LIN {X 0,Y 573.242,Z 122.078,A -85,B 0,C 180,E1 -2301.298,E2 -2301.298} C_VEL
LIN {X 0,Y 573.212,Z 122.081,A -85,B 0,C 180,E1 -2304.018,E2 -2304.018} C_VEL
LIN {X 0,Y 573.238,Z 122.074,A -85,B 0,C 180,E1 -2306.515,E2 -2306.515} C_VEL
LIN {X 0,Y 573.224,Z 122.08,A -85,B 0,C 180,E1 -2309.118,E2 -2309.118} C_VEL
LIN {X 0,Y 573.251,Z 122.075,A -85,B 0,C 180,E1 -2311.971,E2 -2311.971} C_VEL
LIN {X 0,Y 573.252,Z 122.073,A -85,B 0,C 180,E1 -2314.589,E2 -2314.589} C_VEL
LIN {X 0,Y 573.236,Z 122.079,A -85,B 0,C 180,E1 -2317.662,E2 -2317.662} C_VEL
LIN {X 0,Y 573.265,Z 122.073,A -85,B 0,C 180,E1 -2320.67,E2 -2320.67} C_VEL
LIN {X 0,Y 573.246,Z 122.076,A -85,B 0,C 180,E1 -2323.621,E2 -2323.621} C_VEL
LIN {X 0,Y 573.272,Z 122.071,A -85,B 0,C 180,E1 -2325.807,E2 -2325.807} C_VEL
LIN {X 0,Y 573.262,Z 122.076,A -85,B 0,C 180,E1 -2328.745,E2 -2328.745} C_VEL
LIN {X 0,Y 573.281,Z 122.071,A -85,B 0,C 180,E1 -2331.54,E2 -2331.54} C_VEL
LIN {X 0,Y 573.298,Z 122.069,A -85,B 0,C 180,E1 -2334.372,E2 -2334.372} C_VEL
LIN {X 0,Y 573.313,Z 122.065,A -85,B 0,C 180,E1 -2337.892,E2 -2337.892} C_VEL
LIN {X 0,Y 573.334,Z 122.07,A -85,B 0,C 180,E1 -2340.702,E2 -2340.702} C_VEL
LIN {X 0,Y 573.305,Z 122.076,A -85,B 0,C 180,E1 -2342.81,E2 -2342.81} C_VEL
LIN {X 0,Y 573.294,Z 122.067,A -85,B 0,C 180,E1 -2345.628,E2 -2345.628} C_VEL
LIN {X 0,Y 573.289,Z 122.074,A -85,B 0,C 180,E1 -2348.459,E2 -2348.459} C_VEL
LIN {X 0,Y 573.27,Z 122.071,A -85,B 0,C 180,E1 -2351.312,E2 -2351.312} C_VEL
LIN {X 0,Y 573.27,Z 122.074,A -85,B 0,C 180,E1 -2354.193,E2 -2354.193} C_VEL
LIN {X 0,Y 573.256,Z 122.074,A -85,B 0,C 180,E1 -2357.111,E2 -2357.111} C_VEL
LIN {X 0,Y 573.25,Z 122.077,A -85,B 0,C 180,E1 -2360.076,E2 -2360.076} C_VEL
LIN {X 0,Y 573.231,Z 122.076,A -85,B 0,C 180,E1 -2363.099,E2 -2363.099} C_VEL
LIN {X 0,Y 573.247,Z 122.076,A -85,B 0,C 180,E1 -2364.39,E2 -2364.39} C_VEL
LIN {X 0,Y 572.622,Z 122.156,A -85,B 0,C 180,E1 -2364.976,E2 -2364.976} C_VEL
LIN {X 0,Y 569.783,Z 122.509,A -85,B 0,C 180,E1 -2365.928,E2 -2365.928} C_VEL
LIN {X 0,Y 567.355,Z 122.811,A -85,B 0,C 180,E1 -2366.694,E2 -2366.694} C_VEL
LIN {X 0,Y 566.303,Z 122.939,A -85,B 0,C 180,E1 -2367.285,E2 -2367.285} C_VEL
LIN {X 0,Y 566.214,Z 122.95,A -85,B 0,C 180,E1 -2367.485,E2 -2367.485} C_VEL
LIN {X 0,Y 566.184,Z 122.957,A -85,B 0,C 180,E1 -2370.592,E2 -2370.592} C_VEL
LIN {X 0,Y 566.225,Z 122.948,A -85,B 0,C 180,E1 -2373.101,E2 -2373.101} C_VEL
LIN {X 0,Y 566.211,Z 122.958,A -85,B 0,C 180,E1 -2376.216,E2 -2376.216} C_VEL
LIN {X 0,Y 566.219,Z 122.949,A -85,B 0,C 180,E1 -2379.273,E2 -2379.273} C_VEL
LIN {X 0,Y 566.21,Z 122.958,A -85,B 0,C 180,E1 -2382.087,E2 -2382.087} C_VEL
LIN {X 0,Y 566.169,Z 122.955,A -85,B 0,C 180,E1 -2385.036,E2 -2385.036} C_VEL
LIN {X 0,Y 566.21,Z 122.959,A -85,B 0,C 180,E1 -2387.913,E2 -2387.913} C_VEL
LIN {X 0,Y 566.218,Z 122.949,A -85,B 0,C 180,E1 -2390.727,E2 -2390.727} C_VEL
LIN {X 0,Y 566.202,Z 122.96,A -85,B 0,C 180,E1 -2393.785,E2 -2393.785} C_VEL
LIN {X 0,Y 566.225,Z 122.948,A -85,B 0,C 180,E1 -2396.899,E2 -2396.899} C_VEL
LIN {X 0,Y 566.184,Z 122.959,A -85,B 0,C 180,E1 -2399.408,E2 -2399.408} C_VEL
LIN {X 0,Y 566.224,Z 122.953,A -85,B 0,C 180,E1 -2401.858,E2 -2401.858} C_VEL
LIN {X 0,Y 566.211,Z 122.95,A -85,B 0,C 180,E1 -2404.251,E2 -2404.251} C_VEL
LIN {X 0,Y 566.187,Z 122.953,A -85,B 0,C 180,E1 -2406.714,E2 -2406.714} C_VEL
LIN {X 0,Y 566.214,Z 122.955,A -85,B 0,C 180,E1 -2409.663,E2 -2409.663} C_VEL
LIN {X 0,Y 566.196,Z 122.953,A -85,B 0,C 180,E1 -2412.669,E2 -2412.669} C_VEL
LIN {X 0,Y 566.23,Z 122.952,A -85,B 0,C 180,E1 -2415.627,E2 -2415.627} C_VEL
LIN {X 0,Y 566.231,Z 122.949,A -85,B 0,C 180,E1 -2418.675,E2 -2418.675} C_VEL
LIN {X 0,Y 566.23,Z 122.953,A -85,B 0,C 180,E1 -2421.435,E2 -2421.435} C_VEL
LIN {X 0,Y 566.266,Z 122.943,A -85,B 0,C 180,E1 -2424.302,E2 -2424.302} C_VEL
LIN {X 0,Y 566.284,Z 122.941,A -85,B 0,C 180,E1 -2427.867,E2 -2427.867} C_VEL
LIN {X 0,Y 566.3,Z 122.944,A -85,B 0,C 180,E1 -2430.711,E2 -2430.711} C_VEL
LIN {X 0,Y 566.269,Z 122.951,A -85,B 0,C 180,E1 -2432.846,E2 -2432.846} C_VEL
LIN {X 0,Y 566.266,Z 122.943,A -85,B 0,C 180,E1 -2435.699,E2 -2435.699} C_VEL
LIN {X 0,Y 566.231,Z 122.953,A -85,B 0,C 180,E1 -2438.566,E2 -2438.566} C_VEL
LIN {X 0,Y 566.24,Z 122.947,A -85,B 0,C 180,E1 -2441.455,E2 -2441.455} C_VEL
LIN {X 0,Y 566.232,Z 122.954,A -85,B 0,C 180,E1 -2444.507,E2 -2444.507} C_VEL
LIN {X 0,Y 566.198,Z 122.954,A -85,B 0,C 180,E1 -2447.332,E2 -2447.332} C_VEL
LIN {X 0,Y 566.25,Z 123.012,A -85,B 0,C 180,E1 -2449.58,E2 -2449.58} C_VEL
LIN {X 0,Y 566.372,Z 130.978,A -85,B 0,C 180,E1 -2451.092,E2 -2451.092} C_VEL
LIN {X 0,Y 566.202,Z 146.316,A -85,B 0,C 180,E1 -2453.986,E2 -2453.986} C_VEL
LIN {X 0,Y 566.206,Z 146.814,A -85,B 0,C 180,E1 -2454.059,E2 -2454.059} C_VEL
LIN {X 0,Y 567.163,Z 152.949,A -85,B 0,C 180,E1 -2454.162,E2 -2454.162} C_VEL
LIN {X 0,Y 566.894,Z 252.832,A -85,B 0,C 180,E1 -2455.444,E2 -2455.444} C_VEL
LIN {X 0,Y 566.795,Z 265.643,A -85,B 0,C 180,E1 -2455.746,E2 -2455.746} C_VEL
LIN {X 0,Y 566.703,Z 277.817,A -85,B 0,C 180,E1 -2456.17,E2 -2456.17} C_VEL
LIN {X 0,Y 566.583,Z 289.848,A -85,B 0,C 180,E1 -2456.736,E2 -2456.736} C_VEL
LIN {X 0,Y 566.426,Z 301.178,A -85,B 0,C 180,E1 -2457.428,E2 -2457.428} C_VEL
LIN {X 0,Y 566.334,Z 311.622,A -85,B 0,C 180,E1 -2458.228,E2 -2458.228} C_VEL
LIN {X 0,Y 566.205,Z 321.479,A -85,B 0,C 180,E1 -2459.156,E2 -2459.156} C_VEL
LIN {X 0,Y 566.095,Z 330.26,A -85,B 0,C 180,E1 -2460.186,E2 -2460.186} C_VEL
LIN {X 0,Y 566,Z 337.394,A -85,B 0,C 180,E1 -2461.215,E2 -2461.215} C_VEL
LIN {X 0,Y 565.947,Z 343.913,A -85,B 0,C 180,E1 -2462.39,E2 -2462.39} C_VEL
LIN {X 0,Y 565.92,Z 349.394,A -85,B 0,C 180,E1 -2463.691,E2 -2463.691} C_VEL
LIN {X 0,Y 565.868,Z 353.186,A -85,B 0,C 180,E1 -2464.945,E2 -2464.945} C_VEL
LIN {X 0,Y 565.821,Z 355.596,A -85,B 0,C 180,E1 -2466.162,E2 -2466.162} C_VEL
LIN {X 0,Y 565.83,Z 356.879,A -85,B 0,C 180,E1 -2467.49,E2 -2467.49} C_VEL
LIN {X 0,Y 565.816,Z 356.903,A -85,B 0,C 180,E1 -2468.509,E2 -2468.509} C_VEL
LIN {X 0,Y 565.85,Z 355.988,A -85,B 0,C 180,E1 -2469.642,E2 -2469.642} C_VEL
LIN {X 0,Y 565.841,Z 354.118,A -85,B 0,C 180,E1 -2470.744,E2 -2470.744} C_VEL
LIN {X 0,Y 565.926,Z 350.385,A -85,B 0,C 180,E1 -2472.114,E2 -2472.114} C_VEL
LIN {X 0,Y 565.95,Z 346.758,A -85,B 0,C 180,E1 -2473.079,E2 -2473.079} C_VEL
LIN {X 0,Y 565.98,Z 340.891,A -85,B 0,C 180,E1 -2474.28,E2 -2474.28} C_VEL
LIN {X 0,Y 566.059,Z 333.207,A -85,B 0,C 180,E1 -2475.506,E2 -2475.506} C_VEL
LIN {X 0,Y 566.159,Z 325.381,A -85,B 0,C 180,E1 -2476.504,E2 -2476.504} C_VEL
LIN {X 0,Y 566.246,Z 316.412,A -85,B 0,C 180,E1 -2477.435,E2 -2477.435} C_VEL
LIN {X 0,Y 566.36,Z 306.666,A -85,B 0,C 180,E1 -2478.263,E2 -2478.263} C_VEL
LIN {X 0,Y 566.481,Z 294.972,A -85,B 0,C 180,E1 -2479.063,E2 -2479.063} C_VEL
LIN {X 0,Y 566.653,Z 283.646,A -85,B 0,C 180,E1 -2479.665,E2 -2479.665} C_VEL
LIN {X 0,Y 566.816,Z 271.25,A -85,B 0,C 180,E1 -2480.165,E2 -2480.165} C_VEL
LIN {X 0,Y 566.876,Z 258.268,A -85,B 0,C 180,E1 -2480.536,E2 -2480.536} C_VEL
LIN {X 0,Y 566.932,Z 243.917,A -85,B 0,C 180,E1 -2480.774,E2 -2480.774} C_VEL
LIN {X 0,Y 567.131,Z 152.183,A -85,B 0,C 180,E1 -2481.939,E2 -2481.939} C_VEL
LIN {X 0,Y 566.213,Z 146.679,A -85,B 0,C 180,E1 -2482.035,E2 -2482.035} C_VEL
LIN {X 0,Y 566.371,Z 130.971,A -85,B 0,C 180,E1 -2484.984,E2 -2484.984} C_VEL
LIN {X 0,Y 566.246,Z 122.951,A -85,B 0,C 180,E1 -2486.489,E2 -2486.489} C_VEL
LIN {X 0,Y 566.177,Z 122.964,A -85,B 0,C 180,E1 -2489.408,E2 -2489.408} C_VEL
LIN {X 0,Y 566.197,Z 122.955,A -85,B 0,C 180,E1 -2491.857,E2 -2491.857} C_VEL
LIN {X 0,Y 566.207,Z 122.952,A -85,B 0,C 180,E1 -2494.251,E2 -2494.251} C_VEL
LIN {X 0,Y 566.174,Z 122.961,A -85,B 0,C 180,E1 -2497.369,E2 -2497.369} C_VEL
LIN {X 0,Y 566.206,Z 122.952,A -85,B 0,C 180,E1 -2499.663,E2 -2499.663} C_VEL
LIN {X 0,Y 566.183,Z 122.954,A -85,B 0,C 180,E1 -2501.922,E2 -2501.922} C_VEL
LIN {X 0,Y 566.192,Z 122.954,A -85,B 0,C 180,E1 -2504.153,E2 -2504.153} C_VEL
LIN {X 0,Y 566.179,Z 122.959,A -85,B 0,C 180,E1 -2506.359,E2 -2506.359} C_VEL
LIN {X 0,Y 566.235,Z 122.949,A -85,B 0,C 180,E1 -2509.271,E2 -2509.271} C_VEL
LIN {X 0,Y 566.221,Z 122.954,A -85,B 0,C 180,E1 -2512.153,E2 -2512.153} C_VEL
LIN {X 0,Y 566.26,Z 122.946,A -85,B 0,C 180,E1 -2515.016,E2 -2515.016} C_VEL
LIN {X 0,Y 566.281,Z 122.945,A -85,B 0,C 180,E1 -2517.867,E2 -2517.867} C_VEL
LIN {X 0,Y 566.289,Z 122.945,A -85,B 0,C 180,E1 -2520,E2 -2520} C_VEL
LIN {X 0,Y 566.245,Z 122.946,A -85,B 0,C 180,E1 -2522.846,E2 -2522.846} C_VEL
LIN {X 0,Y 566.237,Z 122.951,A -85,B 0,C 180,E1 -2525.699,E2 -2525.699} C_VEL
LIN {X 0,Y 566.188,Z 122.954,A -85,B 0,C 180,E1 -2528.567,E2 -2528.567} C_VEL
LIN {X 0,Y 566.197,Z 122.954,A -85,B 0,C 180,E1 -2531.456,E2 -2531.456} C_VEL
LIN {X 0,Y 566.179,Z 122.954,A -85,B 0,C 180,E1 -2534.482,E2 -2534.482} C_VEL
LIN {X 0,Y 566.151,Z 122.963,A -85,B 0,C 180,E1 -2537.334,E2 -2537.334} C_VEL
LIN {X 0,Y 566.144,Z 122.958,A -85,B 0,C 180,E1 -2540.34,E2 -2540.34} C_VEL
LIN {X 0,Y 566.136,Z 122.96,A -85,B 0,C 180,E1 -2542.634,E2 -2542.634} C_VEL
LIN {X 0,Y 566.15,Z 122.962,A -85,B 0,C 180,E1 -2545.014,E2 -2545.014} C_VEL
LIN {X 0,Y 566.162,Z 122.964,A -85,B 0,C 180,E1 -2547.342,E2 -2547.342} C_VEL
LIN {X 0,Y 566.151,Z 122.959,A -85,B 0,C 180,E1 -2549.772,E2 -2549.772} C_VEL
LIN {X 0,Y 566.196,Z 122.953,A -85,B 0,C 180,E1 -2552.428,E2 -2552.428} C_VEL
LIN {X 0,Y 566.17,Z 122.964,A -85,B 0,C 180,E1 -2554.987,E2 -2554.987} C_VEL
LIN {X 0,Y 566.195,Z 122.954,A -85,B 0,C 180,E1 -2557.461,E2 -2557.461} C_VEL
LIN {X 0,Y 566.21,Z 122.952,A -85,B 0,C 180,E1 -2560.199,E2 -2560.199} C_VEL
LIN {X 0,Y 566.184,Z 122.957,A -85,B 0,C 180,E1 -2563.056,E2 -2563.056} C_VEL
LIN {X 0,Y 566.162,Z 122.96,A -85,B 0,C 180,E1 -2566.053,E2 -2566.053} C_VEL
LIN {X 0,Y 566.174,Z 122.959,A -85,B 0,C 180,E1 -2568.86,E2 -2568.86} C_VEL
LIN {X 0,Y 566.209,Z 122.951,A -85,B 0,C 180,E1 -2571.443,E2 -2571.443} C_VEL
LIN {X 0,Y 566.154,Z 122.967,A -85,B 0,C 180,E1 -2574.307,E2 -2574.307} C_VEL
LIN {X 0,Y 566.215,Z 122.952,A -85,B 0,C 180,E1 -2576.897,E2 -2576.897} C_VEL
LIN {X 0,Y 566.175,Z 122.957,A -85,B 0,C 180,E1 -2579.406,E2 -2579.406} C_VEL
LIN {X 0,Y 566.196,Z 122.96,A -85,B 0,C 180,E1 -2581.856,E2 -2581.856} C_VEL
LIN {X 0,Y 566.242,Z 122.949,A -85,B 0,C 180,E1 -2585.039,E2 -2585.039} C_VEL
LIN {X 0,Y 566.209,Z 122.987,A -85,B 0,C 180,E1 -2586.063,E2 -2586.063} C_VEL
LIN {X 0,Y 566.986,Z 128.165,A -85,B 0,C 180,E1 -2586.824,E2 -2586.824} C_VEL
LIN {X 0,Y 566.84,Z 147.281,A -85,B 0,C 180,E1 -2589.496,E2 -2589.496} C_VEL
LIN {X 0,Y 566.652,Z 167.696,A -85,B 0,C 180,E1 -2592.31,E2 -2592.31} C_VEL
LIN {X 0,Y 566.44,Z 187.948,A -85,B 0,C 180,E1 -2595.08,E2 -2595.08} C_VEL
LIN {X 0,Y 566.414,Z 194.435,A -85,B 0,C 180,E1 -2595.975,E2 -2595.975} C_VEL
LIN {X 0,Y 567.164,Z 201.205,A -85,B 0,C 180,E1 -2596.094,E2 -2596.094} C_VEL
LIN {X 0,Y 566.939,Z 302.924,A -85,B 0,C 180,E1 -2597.402,E2 -2597.402} C_VEL
LIN {X 0,Y 566.856,Z 316.202,A -85,B 0,C 180,E1 -2597.719,E2 -2597.719} C_VEL
LIN {X 0,Y 566.743,Z 328.367,A -85,B 0,C 180,E1 -2598.148,E2 -2598.148} C_VEL
LIN {X 0,Y 566.604,Z 340.231,A -85,B 0,C 180,E1 -2598.712,E2 -2598.712} C_VEL
LIN {X 0,Y 566.44,Z 352.189,A -85,B 0,C 180,E1 -2599.455,E2 -2599.455} C_VEL
LIN {X 0,Y 566.326,Z 362.599,A -85,B 0,C 180,E1 -2600.265,E2 -2600.265} C_VEL
LIN {X 0,Y 566.207,Z 371.109,A -85,B 0,C 180,E1 -2601.074,E2 -2601.074} C_VEL
LIN {X 0,Y 566.113,Z 378.957,A -85,B 0,C 180,E1 -2601.971,E2 -2601.971} C_VEL
LIN {X 0,Y 566.004,Z 386.62,A -85,B 0,C 180,E1 -2603.046,E2 -2603.046} C_VEL
LIN {X 0,Y 566.004,Z 393.677,A -85,B 0,C 180,E1 -2604.299,E2 -2604.299} C_VEL
LIN {X 0,Y 565.933,Z 398.371,A -85,B 0,C 180,E1 -2605.37,E2 -2605.37} C_VEL
LIN {X 0,Y 565.927,Z 401.957,A -85,B 0,C 180,E1 -2606.44,E2 -2606.44} C_VEL
LIN {X 0,Y 565.878,Z 403.806,A -85,B 0,C 180,E1 -2607.152,E2 -2607.152} C_VEL
LIN {X 0,Y 565.846,Z 406.183,A -85,B 0,C 180,E1 -2608.576,E2 -2608.576} C_VEL
LIN {X 0,Y 565.839,Z 407,A -85,B 0,C 180,E1 -2610,E2 -2610} C_VEL
LIN {X 0,Y 565.846,Z 406.185,A -85,B 0,C 180,E1 -2611.423,E2 -2611.423} C_VEL
LIN {X 0,Y 565.878,Z 403.811,A -85,B 0,C 180,E1 -2612.847,E2 -2612.847} C_VEL
LIN {X 0,Y 565.926,Z 400.897,A -85,B 0,C 180,E1 -2613.916,E2 -2613.916} C_VEL
LIN {X 0,Y 565.878,Z 396.95,A -85,B 0,C 180,E1 -2614.987,E2 -2614.987} C_VEL
LIN {X 0,Y 566.004,Z 391.869,A -85,B 0,C 180,E1 -2616.058,E2 -2616.058} C_VEL
LIN {X 0,Y 566.04,Z 385.47,A -85,B 0,C 180,E1 -2617.132,E2 -2617.132} C_VEL
LIN {X 0,Y 566.133,Z 377.481,A -85,B 0,C 180,E1 -2618.207,E2 -2618.207} C_VEL
LIN {X 0,Y 566.229,Z 369.338,A -85,B 0,C 180,E1 -2619.105,E2 -2619.105} C_VEL
LIN {X 0,Y 566.347,Z 359.403,A -85,B 0,C 180,E1 -2620.004,E2 -2620.004} C_VEL
LIN {X 0,Y 566.535,Z 348.297,A -85,B 0,C 180,E1 -2620.807,E2 -2620.807} C_VEL
LIN {X 0,Y 566.612,Z 337.18,A -85,B 0,C 180,E1 -2621.446,E2 -2621.446} C_VEL
LIN {X 0,Y 566.776,Z 324.988,A -85,B 0,C 180,E1 -2621.987,E2 -2621.987} C_VEL
LIN {X 0,Y 566.914,Z 312.19,A -85,B 0,C 180,E1 -2622.393,E2 -2622.393} C_VEL
LIN {X 0,Y 566.958,Z 298.626,A -85,B 0,C 180,E1 -2622.665,E2 -2622.665} C_VEL
LIN {X 0,Y 567.06,Z 198.957,A -85,B 0,C 180,E1 -2623.937,E2 -2623.937} C_VEL
LIN {X 0,Y 566.42,Z 194.441,A -85,B 0,C 180,E1 -2624.024,E2 -2624.024} C_VEL
LIN {X 0,Y 566.627,Z 171.862,A -85,B 0,C 180,E1 -2627.128,E2 -2627.128} C_VEL
LIN {X 0,Y 566.864,Z 150.201,A -85,B 0,C 180,E1 -2630.123,E2 -2630.123} C_VEL
LIN {X 0,Y 567.105,Z 129.879,A -85,B 0,C 180,E1 -2632.977,E2 -2632.977} C_VEL
LIN {X 0,Y 566.833,Z 125.957,A -85,B 0,C 180,E1 -2633.549,E2 -2633.549} C_VEL
LIN {X 0,Y 566.203,Z 122.96,A -85,B 0,C 180,E1 -2634.034,E2 -2634.034} C_VEL
LIN {X 0,Y 566.202,Z 122.955,A -85,B 0,C 180,E1 -2636.657,E2 -2636.657} C_VEL
LIN {X 0,Y 566.203,Z 122.956,A -85,B 0,C 180,E1 -2639.671,E2 -2639.671} C_VEL
LIN {X 0,Y 566.203,Z 122.954,A -85,B 0,C 180,E1 -2642.429,E2 -2642.429} C_VEL
LIN {X 0,Y 566.18,Z 122.954,A -85,B 0,C 180,E1 -2644.989,E2 -2644.989} C_VEL
LIN {X 0,Y 566.197,Z 122.954,A -85,B 0,C 180,E1 -2647.46,E2 -2647.46} C_VEL
LIN {X 0,Y 566.21,Z 122.954,A -85,B 0,C 180,E1 -2650.198,E2 -2650.198} C_VEL
LIN {X 0,Y 566.2,Z 122.952,A -85,B 0,C 180,E1 -2653.054,E2 -2653.054} C_VEL
LIN {X 0,Y 566.199,Z 122.956,A -85,B 0,C 180,E1 -2656.048,E2 -2656.048} C_VEL
LIN {X 0,Y 566.179,Z 122.954,A -85,B 0,C 180,E1 -2658.86,E2 -2658.86} C_VEL
LIN {X 0,Y 566.186,Z 122.963,A -85,B 0,C 180,E1 -2661.636,E2 -2661.636} C_VEL
LIN {X 0,Y 566.161,Z 122.957,A -85,B 0,C 180,E1 -2664.307,E2 -2664.307} C_VEL
LIN {X 0,Y 566.204,Z 122.952,A -85,B 0,C 180,E1 -2666.896,E2 -2666.896} C_VEL
LIN {X 0,Y 566.175,Z 122.963,A -85,B 0,C 180,E1 -2669.407,E2 -2669.407} C_VEL
LIN {X 0,Y 566.211,Z 122.953,A -85,B 0,C 180,E1 -2671.857,E2 -2671.857} C_VEL
LIN {X 0,Y 566.212,Z 122.95,A -85,B 0,C 180,E1 -2674.251,E2 -2674.251} C_VEL
LIN {X 0,Y 566.171,Z 122.956,A -85,B 0,C 180,E1 -2676.718,E2 -2676.718} C_VEL
LIN {X 0,Y 566.207,Z 122.954,A -85,B 0,C 180,E1 -2679.662,E2 -2679.662} C_VEL
LIN {X 0,Y 566.197,Z 122.954,A -85,B 0,C 180,E1 -2682.668,E2 -2682.668} C_VEL
LIN {X 0,Y 566.233,Z 122.95,A -85,B 0,C 180,E1 -2685.626,E2 -2685.626} C_VEL
LIN {X 0,Y 566.234,Z 122.95,A -85,B 0,C 180,E1 -2688.675,E2 -2688.675} C_VEL
LIN {X 0,Y 566.226,Z 122.951,A -85,B 0,C 180,E1 -2691.434,E2 -2691.434} C_VEL
LIN {X 0,Y 566.266,Z 122.944,A -85,B 0,C 180,E1 -2694.301,E2 -2694.301} C_VEL
LIN {X 0,Y 566.284,Z 122.941,A -85,B 0,C 180,E1 -2697.866,E2 -2697.866} C_VEL
LIN {X 0,Y 566.304,Z 122.946,A -85,B 0,C 180,E1 -2700.711,E2 -2700.711} C_VEL
LIN {X 0,Y 566.271,Z 122.951,A -85,B 0,C 180,E1 -2702.845,E2 -2702.845} C_VEL
LIN {X 0,Y 566.262,Z 122.943,A -85,B 0,C 180,E1 -2705.698,E2 -2705.698} C_VEL
LIN {X 0,Y 566.232,Z 122.955,A -85,B 0,C 180,E1 -2708.565,E2 -2708.565} C_VEL
LIN {X 0,Y 566.24,Z 122.946,A -85,B 0,C 180,E1 -2711.454,E2 -2711.454} C_VEL
LIN {X 0,Y 566.232,Z 122.957,A -85,B 0,C 180,E1 -2714.506,E2 -2714.506} C_VEL
LIN {X 0,Y 566.197,Z 122.952,A -85,B 0,C 180,E1 -2717.331,E2 -2717.331} C_VEL
LIN {X 0,Y 566.211,Z 122.958,A -85,B 0,C 180,E1 -2720.337,E2 -2720.337} C_VEL
LIN {X 0,Y 566.17,Z 122.955,A -85,B 0,C 180,E1 -2723.282,E2 -2723.282} C_VEL
LIN {X 0,Y 566.221,Z 122.95,A -85,B 0,C 180,E1 -2725.748,E2 -2725.748} C_VEL
LIN {X 0,Y 566.214,Z 122.95,A -85,B 0,C 180,E1 -2727.485,E2 -2727.485} C_VEL
LIN {X 0,Y 565.534,Z 123.042,A -85,B 0,C 180,E1 -2728.079,E2 -2728.079} C_VEL
LIN {X 0,Y 562.663,Z 123.4,A -85,B 0,C 180,E1 -2729.043,E2 -2729.043} C_VEL
LIN {X 0,Y 560.249,Z 123.7,A -85,B 0,C 180,E1 -2729.818,E2 -2729.818} C_VEL
LIN {X 0,Y 559.221,Z 123.827,A -85,B 0,C 180,E1 -2730.417,E2 -2730.417} C_VEL
LIN {X 0,Y 559.142,Z 123.833,A -85,B 0,C 180,E1 -2730.619,E2 -2730.619} C_VEL
LIN {X 0,Y 559.161,Z 123.83,A -85,B 0,C 180,E1 -2733.574,E2 -2733.574} C_VEL
LIN {X 0,Y 559.163,Z 123.832,A -85,B 0,C 180,E1 -2736.448,E2 -2736.448} C_VEL
LIN {X 0,Y 559.175,Z 123.826,A -85,B 0,C 180,E1 -2738.933,E2 -2738.933} C_VEL
LIN {X 0,Y 559.188,Z 123.831,A -85,B 0,C 180,E1 -2741.767,E2 -2741.767} C_VEL
LIN {X 0,Y 559.136,Z 123.831,A -85,B 0,C 180,E1 -2744.739,E2 -2744.739} C_VEL
LIN {X 0,Y 559.16,Z 123.83,A -85,B 0,C 180,E1 -2747.257,E2 -2747.257} C_VEL
LIN {X 0,Y 559.182,Z 123.83,A -85,B 0,C 180,E1 -2750.135,E2 -2750.135} C_VEL
LIN {X 0,Y 559.141,Z 123.831,A -85,B 0,C 180,E1 -2752.892,E2 -2752.892} C_VEL
LIN {X 0,Y 559.161,Z 123.832,A -85,B 0,C 180,E1 -2756.051,E2 -2756.051} C_VEL
LIN {X 0,Y 559.159,Z 123.829,A -85,B 0,C 180,E1 -2758.981,E2 -2758.981} C_VEL
LIN {X 0,Y 559.188,Z 123.825,A -85,B 0,C 180,E1 -2762.289,E2 -2762.289} C_VEL
LIN {X 0,Y 559.175,Z 123.827,A -85,B 0,C 180,E1 -2764.813,E2 -2764.813} C_VEL
LIN {X 0,Y 559.138,Z 123.835,A -85,B 0,C 180,E1 -2767.847,E2 -2767.847} C_VEL
LIN {X 0,Y 559.194,Z 123.824,A -85,B 0,C 180,E1 -2770.492,E2 -2770.492} C_VEL
LIN {X 0,Y 559.178,Z 123.833,A -85,B 0,C 180,E1 -2773.198,E2 -2773.198} C_VEL
LIN {X 0,Y 559.169,Z 123.827,A -85,B 0,C 180,E1 -2776.184,E2 -2776.184} C_VEL
LIN {X 0,Y 559.193,Z 123.832,A -85,B 0,C 180,E1 -2779.134,E2 -2779.134} C_VEL
LIN {X 0,Y 559.202,Z 123.823,A -85,B 0,C 180,E1 -2782.054,E2 -2782.054} C_VEL
LIN {X 0,Y 559.253,Z 123.824,A -85,B 0,C 180,E1 -2784.954,E2 -2784.954} C_VEL
LIN {X 0,Y 559.254,Z 123.817,A -85,B 0,C 180,E1 -2787.84,E2 -2787.84} C_VEL
LIN {X 0,Y 559.27,Z 123.82,A -85,B 0,C 180,E1 -2790.72,E2 -2790.72} C_VEL
LIN {X 0,Y 559.236,Z 123.828,A -85,B 0,C 180,E1 -2792.882,E2 -2792.882} C_VEL
LIN {X 0,Y 559.236,Z 123.819,A -85,B 0,C 180,E1 -2795.771,E2 -2795.771} C_VEL
LIN {X 0,Y 559.189,Z 123.832,A -85,B 0,C 180,E1 -2798.675,E2 -2798.675} C_VEL
LIN {X 0,Y 559.203,Z 123.823,A -85,B 0,C 180,E1 -2801.601,E2 -2801.601} C_VEL
LIN {X 0,Y 559.198,Z 123.832,A -85,B 0,C 180,E1 -2804.596,E2 -2804.596} C_VEL
LIN {X 0,Y 559.158,Z 123.83,A -85,B 0,C 180,E1 -2807.557,E2 -2807.557} C_VEL
LIN {X 0,Y 559.248,Z 123.996,A -85,B 0,C 180,E1 -2809.523,E2 -2809.523} C_VEL
LIN {X 0,Y 559.342,Z 133.681,A -85,B 0,C 180,E1 -2811.37,E2 -2811.37} C_VEL
LIN {X 0,Y 559.2,Z 146.846,A -85,B 0,C 180,E1 -2813.862,E2 -2813.862} C_VEL
LIN {X 0,Y 560.299,Z 154.738,A -85,B 0,C 180,E1 -2814.009,E2 -2814.009} C_VEL
LIN {X 0,Y 559.974,Z 252.81,A -85,B 0,C 180,E1 -2815.284,E2 -2815.284} C_VEL
LIN {X 0,Y 559.864,Z 265.998,A -85,B 0,C 180,E1 -2815.599,E2 -2815.599} C_VEL
LIN {X 0,Y 559.725,Z 279.132,A -85,B 0,C 180,E1 -2816.07,E2 -2816.07} C_VEL
LIN {X 0,Y 559.583,Z 291.429,A -85,B 0,C 180,E1 -2816.68,E2 -2816.68} C_VEL
LIN {X 0,Y 559.422,Z 302.19,A -85,B 0,C 180,E1 -2817.365,E2 -2817.365} C_VEL
LIN {X 0,Y 559.275,Z 313.401,A -85,B 0,C 180,E1 -2818.256,E2 -2818.256} C_VEL
LIN {X 0,Y 559.163,Z 322.417,A -85,B 0,C 180,E1 -2819.147,E2 -2819.147} C_VEL
LIN {X 0,Y 559.037,Z 331.034,A -85,B 0,C 180,E1 -2820.19,E2 -2820.19} C_VEL
LIN {X 0,Y 558.922,Z 338.056,A -85,B 0,C 180,E1 -2821.236,E2 -2821.236} C_VEL
LIN {X 0,Y 558.889,Z 343.488,A -85,B 0,C 180,E1 -2822.233,E2 -2822.233} C_VEL
LIN {X 0,Y 558.823,Z 349.268,A -85,B 0,C 180,E1 -2823.599,E2 -2823.599} C_VEL
LIN {X 0,Y 558.799,Z 352.05,A -85,B 0,C 180,E1 -2824.47,E2 -2824.47} C_VEL
LIN {X 0,Y 558.754,Z 354.199,A -85,B 0,C 180,E1 -2825.352,E2 -2825.352} C_VEL
LIN {X 0,Y 558.732,Z 355.945,A -85,B 0,C 180,E1 -2826.388,E2 -2826.388} C_VEL
LIN {X 0,Y 558.741,Z 356.905,A -85,B 0,C 180,E1 -2827.587,E2 -2827.587} C_VEL
LIN {X 0,Y 558.729,Z 356.648,A -85,B 0,C 180,E1 -2828.972,E2 -2828.972} C_VEL
LIN {X 0,Y 558.763,Z 355.67,A -85,B 0,C 180,E1 -2829.902,E2 -2829.902} C_VEL
LIN {X 0,Y 558.758,Z 353.628,A -85,B 0,C 180,E1 -2831.004,E2 -2831.004} C_VEL
LIN {X 0,Y 558.836,Z 349.543,A -85,B 0,C 180,E1 -2832.411,E2 -2832.411} C_VEL
LIN {X 0,Y 558.848,Z 345.445,A -85,B 0,C 180,E1 -2833.439,E2 -2833.439} C_VEL
LIN {X 0,Y 558.916,Z 340.328,A -85,B 0,C 180,E1 -2834.46,E2 -2834.46} C_VEL
LIN {X 0,Y 559.01,Z 332.628,A -85,B 0,C 180,E1 -2835.685,E2 -2835.685} C_VEL
LIN {X 0,Y 559.135,Z 323.65,A -85,B 0,C 180,E1 -2836.806,E2 -2836.806} C_VEL
LIN {X 0,Y 559.262,Z 314.305,A -85,B 0,C 180,E1 -2837.751,E2 -2837.751} C_VEL
LIN {X 0,Y 559.404,Z 303.73,A -85,B 0,C 180,E1 -2838.616,E2 -2838.616} C_VEL
LIN {X 0,Y 559.546,Z 292.912,A -85,B 0,C 180,E1 -2839.325,E2 -2839.325} C_VEL
LIN {X 0,Y 559.735,Z 281.309,A -85,B 0,C 180,E1 -2839.923,E2 -2839.923} C_VEL
LIN {X 0,Y 559.88,Z 269.862,A -85,B 0,C 180,E1 -2840.37,E2 -2840.37} C_VEL
LIN {X 0,Y 559.966,Z 257.444,A -85,B 0,C 180,E1 -2840.713,E2 -2840.713} C_VEL
LIN {X 0,Y 560.053,Z 241.005,A -85,B 0,C 180,E1 -2840.972,E2 -2840.972} C_VEL
LIN {X 0,Y 560.276,Z 153.238,A -85,B 0,C 180,E1 -2842.101,E2 -2842.101} C_VEL
LIN {X 0,Y 559.229,Z 146.915,A -85,B 0,C 180,E1 -2842.22,E2 -2842.22} C_VEL
LIN {X 0,Y 559.367,Z 131.224,A -85,B 0,C 180,E1 -2845.165,E2 -2845.165} C_VEL
LIN {X 0,Y 559.215,Z 123.828,A -85,B 0,C 180,E1 -2846.564,E2 -2846.564} C_VEL
LIN {X 0,Y 559.154,Z 123.835,A -85,B 0,C 180,E1 -2848.981,E2 -2848.981} C_VEL
LIN {X 0,Y 559.171,Z 123.833,A -85,B 0,C 180,E1 -2851.62,E2 -2851.62} C_VEL
LIN {X 0,Y 559.178,Z 123.829,A -85,B 0,C 180,E1 -2853.903,E2 -2853.903} C_VEL
LIN {X 0,Y 559.119,Z 123.844,A -85,B 0,C 180,E1 -2857.067,E2 -2857.067} C_VEL
LIN {X 0,Y 559.176,Z 123.831,A -85,B 0,C 180,E1 -2859.396,E2 -2859.396} C_VEL
LIN {X 0,Y 559.132,Z 123.833,A -85,B 0,C 180,E1 -2861.686,E2 -2861.686} C_VEL
LIN {X 0,Y 559.156,Z 123.83,A -85,B 0,C 180,E1 -2863.948,E2 -2863.948} C_VEL
LIN {X 0,Y 559.156,Z 123.832,A -85,B 0,C 180,E1 -2866.184,E2 -2866.184} C_VEL
LIN {X 0,Y 559.194,Z 123.827,A -85,B 0,C 180,E1 -2869.134,E2 -2869.134} C_VEL
LIN {X 0,Y 559.192,Z 123.828,A -85,B 0,C 180,E1 -2872.054,E2 -2872.054} C_VEL
LIN {X 0,Y 559.236,Z 123.821,A -85,B 0,C 180,E1 -2874.954,E2 -2874.954} C_VEL
LIN {X 0,Y 559.252,Z 123.82,A -85,B 0,C 180,E1 -2877.84,E2 -2877.84} C_VEL
LIN {X 0,Y 559.258,Z 123.821,A -85,B 0,C 180,E1 -2880,E2 -2880} C_VEL
LIN {X 0,Y 559.212,Z 123.821,A -85,B 0,C 180,E1 -2882.882,E2 -2882.882} C_VEL
LIN {X 0,Y 559.207,Z 123.828,A -85,B 0,C 180,E1 -2885.771,E2 -2885.771} C_VEL
LIN {X 0,Y 559.153,Z 123.83,A -85,B 0,C 180,E1 -2888.675,E2 -2888.675} C_VEL
LIN {X 0,Y 559.158,Z 123.833,A -85,B 0,C 180,E1 -2891.602,E2 -2891.602} C_VEL
LIN {X 0,Y 559.138,Z 123.83,A -85,B 0,C 180,E1 -2894.568,E2 -2894.568} C_VEL
LIN {X 0,Y 559.107,Z 123.844,A -85,B 0,C 180,E1 -2897.559,E2 -2897.559} C_VEL
LIN {X 0,Y 559.106,Z 123.835,A -85,B 0,C 180,E1 -2900.608,E2 -2900.608} C_VEL
LIN {X 0,Y 559.107,Z 123.839,A -85,B 0,C 180,E1 -2903.719,E2 -2903.719} C_VEL
LIN {X 0,Y 559.146,Z 123.831,A -85,B 0,C 180,E1 -2906.099,E2 -2906.099} C_VEL
LIN {X 0,Y 559.103,Z 123.836,A -85,B 0,C 180,E1 -2908.533,E2 -2908.533} C_VEL
LIN {X 0,Y 559.125,Z 123.839,A -85,B 0,C 180,E1 -2911.269,E2 -2911.269} C_VEL
LIN {X 0,Y 559.157,Z 123.829,A -85,B 0,C 180,E1 -2913.947,E2 -2913.947} C_VEL
LIN {X 0,Y 559.135,Z 123.837,A -85,B 0,C 180,E1 -2917.109,E2 -2917.109} C_VEL
LIN {X 0,Y 559.16,Z 123.829,A -85,B 0,C 180,E1 -2919.941,E2 -2919.941} C_VEL
LIN {X 0,Y 559.146,Z 123.839,A -85,B 0,C 180,E1 -2922.745,E2 -2922.745} C_VEL
LIN {X 0,Y 559.128,Z 123.834,A -85,B 0,C 180,E1 -2925.764,E2 -2925.764} C_VEL
LIN {X 0,Y 559.158,Z 123.835,A -85,B 0,C 180,E1 -2928.229,E2 -2928.229} C_VEL
LIN {X 0,Y 559.175,Z 123.828,A -85,B 0,C 180,E1 -2931.192,E2 -2931.192} C_VEL
LIN {X 0,Y 559.126,Z 123.836,A -85,B 0,C 180,E1 -2933.788,E2 -2933.788} C_VEL
LIN {X 0,Y 559.165,Z 123.836,A -85,B 0,C 180,E1 -2936.425,E2 -2936.425} C_VEL
LIN {X 0,Y 559.154,Z 123.831,A -85,B 0,C 180,E1 -2938.98,E2 -2938.98} C_VEL
LIN {X 0,Y 559.149,Z 123.835,A -85,B 0,C 180,E1 -2941.623,E2 -2941.623} C_VEL
LIN {X 0,Y 559.168,Z 123.837,A -85,B 0,C 180,E1 -2943.902,E2 -2943.902} C_VEL
LIN {X 0,Y 559.202,Z 123.954,A -85,B 0,C 180,E1 -2945.941,E2 -2945.941} C_VEL
LIN {X 0,Y 560.053,Z 129.313,A -85,B 0,C 180,E1 -2946.739,E2 -2946.739} C_VEL
LIN {X 0,Y 559.853,Z 148.267,A -85,B 0,C 180,E1 -2949.421,E2 -2949.421} C_VEL
LIN {X 0,Y 559.601,Z 170.031,A -85,B 0,C 180,E1 -2952.457,E2 -2952.457} C_VEL
LIN {X 0,Y 559.416,Z 187.656,A -85,B 0,C 180,E1 -2954.889,E2 -2954.889} C_VEL
LIN {X 0,Y 559.416,Z 194.254,A -85,B 0,C 180,E1 -2955.796,E2 -2955.796} C_VEL
LIN {X 0,Y 560.282,Z 202.068,A -85,B 0,C 180,E1 -2955.934,E2 -2955.934} C_VEL
LIN {X 0,Y 560.04,Z 302.922,A -85,B 0,C 180,E1 -2957.244,E2 -2957.244} C_VEL
LIN {X 0,Y 559.914,Z 316.202,A -85,B 0,C 180,E1 -2957.564,E2 -2957.564} C_VEL
LIN {X 0,Y 559.78,Z 329.487,A -85,B 0,C 180,E1 -2958.044,E2 -2958.044} C_VEL
LIN {X 0,Y 559.605,Z 341.921,A -85,B 0,C 180,E1 -2958.667,E2 -2958.667} C_VEL
LIN {X 0,Y 559.427,Z 353.478,A -85,B 0,C 180,E1 -2959.412,E2 -2959.412} C_VEL
LIN {X 0,Y 559.297,Z 363.641,A -85,B 0,C 180,E1 -2960.233,E2 -2960.233} C_VEL
LIN {X 0,Y 559.135,Z 372.782,A -85,B 0,C 180,E1 -2961.142,E2 -2961.142} C_VEL
LIN {X 0,Y 559.01,Z 381.685,A -85,B 0,C 180,E1 -2962.232,E2 -2962.232} C_VEL
LIN {X 0,Y 558.926,Z 387.737,A -85,B 0,C 180,E1 -2963.139,E2 -2963.139} C_VEL
LIN {X 0,Y 558.936,Z 393.677,A -85,B 0,C 180,E1 -2964.226,E2 -2964.226} C_VEL
LIN {X 0,Y 558.827,Z 398.371,A -85,B 0,C 180,E1 -2965.311,E2 -2965.311} C_VEL
LIN {X 0,Y 558.836,Z 401.957,A -85,B 0,C 180,E1 -2966.394,E2 -2966.394} C_VEL
LIN {X 0,Y 558.799,Z 403.806,A -85,B 0,C 180,E1 -2967.116,E2 -2967.116} C_VEL
LIN {X 0,Y 558.745,Z 406.182,A -85,B 0,C 180,E1 -2968.558,E2 -2968.558} C_VEL
LIN {X 0,Y 558.74,Z 407,A -85,B 0,C 180,E1 -2970,E2 -2970} C_VEL
LIN {X 0,Y 558.745,Z 406.185,A -85,B 0,C 180,E1 -2971.441,E2 -2971.441} C_VEL
LIN {X 0,Y 558.799,Z 403.811,A -85,B 0,C 180,E1 -2972.883,E2 -2972.883} C_VEL
LIN {X 0,Y 558.844,Z 400.897,A -85,B 0,C 180,E1 -2973.966,E2 -2973.966} C_VEL
LIN {X 0,Y 558.798,Z 396.95,A -85,B 0,C 180,E1 -2975.05,E2 -2975.05} C_VEL
LIN {X 0,Y 558.92,Z 391.869,A -85,B 0,C 180,E1 -2976.135,E2 -2976.135} C_VEL
LIN {X 0,Y 558.977,Z 385.469,A -85,B 0,C 180,E1 -2977.222,E2 -2977.222} C_VEL
LIN {X 0,Y 559.099,Z 377.48,A -85,B 0,C 180,E1 -2978.311,E2 -2978.311} C_VEL
LIN {X 0,Y 559.194,Z 369.337,A -85,B 0,C 180,E1 -2979.221,E2 -2979.221} C_VEL
LIN {X 0,Y 559.357,Z 359.402,A -85,B 0,C 180,E1 -2980.131,E2 -2980.131} C_VEL
LIN {X 0,Y 559.556,Z 348.403,A -85,B 0,C 180,E1 -2980.936,E2 -2980.936} C_VEL
LIN {X 0,Y 559.671,Z 336.464,A -85,B 0,C 180,E1 -2981.627,E2 -2981.627} C_VEL
LIN {X 0,Y 559.82,Z 324.986,A -85,B 0,C 180,E1 -2982.138,E2 -2982.138} C_VEL
LIN {X 0,Y 559.968,Z 312.189,A -85,B 0,C 180,E1 -2982.549,E2 -2982.549} C_VEL
LIN {X 0,Y 560.057,Z 298.617,A -85,B 0,C 180,E1 -2982.823,E2 -2982.823} C_VEL
LIN {X 0,Y 560.223,Z 200.12,A -85,B 0,C 180,E1 -2984.093,E2 -2984.093} C_VEL
LIN {X 0,Y 559.412,Z 194.301,A -85,B 0,C 180,E1 -2984.204,E2 -2984.204} C_VEL
LIN {X 0,Y 559.62,Z 172.338,A -85,B 0,C 180,E1 -2987.243,E2 -2987.243} C_VEL
LIN {X 0,Y 559.876,Z 151.267,A -85,B 0,C 180,E1 -2990.194,E2 -2990.194} C_VEL
LIN {X 0,Y 560.189,Z 131.019,A -85,B 0,C 180,E1 -2993.075,E2 -2993.075} C_VEL
LIN {X 0,Y 559.513,Z 125.543,A -85,B 0,C 180,E1 -2993.896,E2 -2993.896} C_VEL
LIN {X 0,Y 559.164,Z 123.837,A -85,B 0,C 180,E1 -2994.183,E2 -2994.183} C_VEL
LIN {X 0,Y 559.165,Z 123.83,A -85,B 0,C 180,E1 -2996.902,E2 -2996.902} C_VEL
LIN {X 0,Y 559.149,Z 123.837,A -85,B 0,C 180,E1 -2999.857,E2 -2999.857} C_VEL
LIN {X 0,Y 559.157,Z 123.829,A -85,B 0,C 180,E1 -3002.715,E2 -3002.715} C_VEL
LIN {X 0,Y 559.128,Z 123.833,A -85,B 0,C 180,E1 -3005.324,E2 -3005.324} C_VEL
LIN {X 0,Y 559.134,Z 123.839,A -85,B 0,C 180,E1 -3008.017,E2 -3008.017} C_VEL
LIN {X 0,Y 559.156,Z 123.829,A -85,B 0,C 180,E1 -3010.812,E2 -3010.812} C_VEL
LIN {X 0,Y 559.139,Z 123.84,A -85,B 0,C 180,E1 -3013.734,E2 -3013.734} C_VEL
LIN {X 0,Y 559.147,Z 123.83,A -85,B 0,C 180,E1 -3016.803,E2 -3016.803} C_VEL
LIN {X 0,Y 559.158,Z 123.831,A -85,B 0,C 180,E1 -3019.187,E2 -3019.187} C_VEL
LIN {X 0,Y 559.133,Z 123.836,A -85,B 0,C 180,E1 -3021.982,E2 -3021.982} C_VEL
LIN {X 0,Y 559.13,Z 123.832,A -85,B 0,C 180,E1 -3024.787,E2 -3024.787} C_VEL
LIN {X 0,Y 559.154,Z 123.836,A -85,B 0,C 180,E1 -3027.364,E2 -3027.364} C_VEL
LIN {X 0,Y 559.144,Z 123.831,A -85,B 0,C 180,E1 -3030.143,E2 -3030.143} C_VEL
LIN {X 0,Y 559.169,Z 123.832,A -85,B 0,C 180,E1 -3033.097,E2 -3033.097} C_VEL
LIN {X 0,Y 559.155,Z 123.836,A -85,B 0,C 180,E1 -3035.494,E2 -3035.494} C_VEL
LIN {X 0,Y 559.171,Z 123.828,A -85,B 0,C 180,E1 -3038.623,E2 -3038.623} C_VEL
LIN {X 0,Y 559.16,Z 123.833,A -85,B 0,C 180,E1 -3040.926,E2 -3040.926} C_VEL
LIN {X 0,Y 559.163,Z 123.828,A -85,B 0,C 180,E1 -3043.947,E2 -3043.947} C_VEL
LIN {X 0,Y 559.171,Z 123.827,A -85,B 0,C 180,E1 -3046.184,E2 -3046.184} C_VEL
LIN {X 0,Y 559.194,Z 123.833,A -85,B 0,C 180,E1 -3049.133,E2 -3049.133} C_VEL
LIN {X 0,Y 559.203,Z 123.823,A -85,B 0,C 180,E1 -3052.053,E2 -3052.053} C_VEL
LIN {X 0,Y 559.252,Z 123.827,A -85,B 0,C 180,E1 -3054.953,E2 -3054.953} C_VEL
LIN {X 0,Y 559.254,Z 123.816,A -85,B 0,C 180,E1 -3057.839,E2 -3057.839} C_VEL
LIN {X 0,Y 559.274,Z 123.822,A -85,B 0,C 180,E1 -3060.72,E2 -3060.72} C_VEL
LIN {X 0,Y 559.237,Z 123.827,A -85,B 0,C 180,E1 -3062.881,E2 -3062.881} C_VEL
LIN {X 0,Y 559.231,Z 123.819,A -85,B 0,C 180,E1 -3065.77,E2 -3065.77} C_VEL
LIN {X 0,Y 559.19,Z 123.834,A -85,B 0,C 180,E1 -3068.674,E2 -3068.674} C_VEL
LIN {X 0,Y 559.203,Z 123.823,A -85,B 0,C 180,E1 -3071.6,E2 -3071.6} C_VEL
LIN {X 0,Y 559.197,Z 123.833,A -85,B 0,C 180,E1 -3074.595,E2 -3074.595} C_VEL
LIN {X 0,Y 559.157,Z 123.828,A -85,B 0,C 180,E1 -3077.557,E2 -3077.557} C_VEL
LIN {X 0,Y 559.17,Z 123.828,A -85,B 0,C 180,E1 -3079.837,E2 -3079.837} C_VEL
LIN {X 0,Y 559.139,Z 123.837,A -85,B 0,C 180,E1 -3082.152,E2 -3082.152} C_VEL
LIN {X 0,Y 559.175,Z 123.826,A -85,B 0,C 180,E1 -3085.298,E2 -3085.298} C_VEL
LIN {X 0,Y 559.192,Z 123.826,A -85,B 0,C 180,E1 -3087.711,E2 -3087.711} C_VEL
LIN {X 0,Y 559.142,Z 123.833,A -85,B 0,C 180,E1 -3090.619,E2 -3090.619} C_VEL
LIN {X 0,Y 558.482,Z 123.915,A -85,B 0,C 180,E1 -3091.221,E2 -3091.221} C_VEL
LIN {X 0,Y 555.621,Z 124.279,A -85,B 0,C 180,E1 -3092.197,E2 -3092.197} C_VEL
LIN {X 0,Y 553.207,Z 124.574,A -85,B 0,C 180,E1 -3092.983,E2 -3092.983} C_VEL
LIN {X 0,Y 552.184,Z 124.699,A -85,B 0,C 180,E1 -3093.589,E2 -3093.589} C_VEL
LIN {X 0,Y 552.109,Z 124.711,A -85,B 0,C 180,E1 -3093.795,E2 -3093.795} C_VEL
LIN {X 0,Y 552.107,Z 124.708,A -85,B 0,C 180,E1 -3096.746,E2 -3096.746} C_VEL
LIN {X 0,Y 552.131,Z 124.706,A -85,B 0,C 180,E1 -3099.526,E2 -3099.526} C_VEL
LIN {X 0,Y 552.126,Z 124.707,A -85,B 0,C 180,E1 -3102.425,E2 -3102.425} C_VEL
LIN {X 0,Y 552.095,Z 124.712,A -85,B 0,C 180,E1 -3105.563,E2 -3105.563} C_VEL
LIN {X 0,Y 552.136,Z 124.703,A -85,B 0,C 180,E1 -3108.676,E2 -3108.676} C_VEL
LIN {X 0,Y 552.116,Z 124.709,A -85,B 0,C 180,E1 -3111.411,E2 -3111.411} C_VEL
LIN {X 0,Y 552.098,Z 124.711,A -85,B 0,C 180,E1 -3114.158,E2 -3114.158} C_VEL
LIN {X 0,Y 552.119,Z 124.705,A -85,B 0,C 180,E1 -3116.815,E2 -3116.815} C_VEL
LIN {X 0,Y 552.103,Z 124.713,A -85,B 0,C 180,E1 -3119.391,E2 -3119.391} C_VEL
LIN {X 0,Y 552.122,Z 124.709,A -85,B 0,C 180,E1 -3121.903,E2 -3121.903} C_VEL
LIN {X 0,Y 552.151,Z 124.701,A -85,B 0,C 180,E1 -3124.65,E2 -3124.65} C_VEL
LIN {X 0,Y 552.092,Z 124.717,A -85,B 0,C 180,E1 -3127.549,E2 -3127.549} C_VEL
LIN {X 0,Y 552.146,Z 124.702,A -85,B 0,C 180,E1 -3130.373,E2 -3130.373} C_VEL
LIN {X 0,Y 552.152,Z 124.705,A -85,B 0,C 180,E1 -3132.978,E2 -3132.978} C_VEL
LIN {X 0,Y 552.132,Z 124.704,A -85,B 0,C 180,E1 -3136.005,E2 -3136.005} C_VEL
LIN {X 0,Y 552.16,Z 124.706,A -85,B 0,C 180,E1 -3138.994,E2 -3138.994} C_VEL
LIN {X 0,Y 552.156,Z 124.701,A -85,B 0,C 180,E1 -3141.952,E2 -3141.952} C_VEL
LIN {X 0,Y 552.228,Z 124.698,A -85,B 0,C 180,E1 -3144.889,E2 -3144.889} C_VEL
LIN {X 0,Y 552.225,Z 124.692,A -85,B 0,C 180,E1 -3147.812,E2 -3147.812} C_VEL
LIN {X 0,Y 552.24,Z 124.696,A -85,B 0,C 180,E1 -3150.73,E2 -3150.73} C_VEL
LIN {X 0,Y 552.202,Z 124.704,A -85,B 0,C 180,E1 -3152.919,E2 -3152.919} C_VEL
LIN {X 0,Y 552.207,Z 124.694,A -85,B 0,C 180,E1 -3155.844,E2 -3155.844} C_VEL
LIN {X 0,Y 552.16,Z 124.709,A -85,B 0,C 180,E1 -3158.786,E2 -3158.786} C_VEL
LIN {X 0,Y 552.161,Z 124.7,A -85,B 0,C 180,E1 -3161.751,E2 -3161.751} C_VEL
LIN {X 0,Y 552.135,Z 124.713,A -85,B 0,C 180,E1 -3164.749,E2 -3164.749} C_VEL
LIN {X 0,Y 552.11,Z 124.709,A -85,B 0,C 180,E1 -3167.789,E2 -3167.789} C_VEL
LIN {X 0,Y 552.194,Z 124.859,A -85,B 0,C 180,E1 -3169.435,E2 -3169.435} C_VEL
LIN {X 0,Y 552.377,Z 132.328,A -85,B 0,C 180,E1 -3170.871,E2 -3170.871} C_VEL
LIN {X 0,Y 552.217,Z 147.218,A -85,B 0,C 180,E1 -3173.697,E2 -3173.697} C_VEL
LIN {X 0,Y 553.428,Z 155.026,A -85,B 0,C 180,E1 -3173.832,E2 -3173.832} C_VEL
LIN {X 0,Y 553.062,Z 254.08,A -85,B 0,C 180,E1 -3175.145,E2 -3175.145} C_VEL
LIN {X 0,Y 552.952,Z 267.752,A -85,B 0,C 180,E1 -3175.489,E2 -3175.489} C_VEL
LIN {X 0,Y 552.805,Z 280.441,A -85,B 0,C 180,E1 -3175.965,E2 -3175.965} C_VEL
LIN {X 0,Y 552.66,Z 291.475,A -85,B 0,C 180,E1 -3176.523,E2 -3176.523} C_VEL
LIN {X 0,Y 552.441,Z 302.858,A -85,B 0,C 180,E1 -3177.257,E2 -3177.257} C_VEL
LIN {X 0,Y 552.284,Z 313.175,A -85,B 0,C 180,E1 -3178.089,E2 -3178.089} C_VEL
LIN {X 0,Y 552.134,Z 321.677,A -85,B 0,C 180,E1 -3178.927,E2 -3178.927} C_VEL
LIN {X 0,Y 551.995,Z 330.747,A -85,B 0,C 180,E1 -3180.03,E2 -3180.03} C_VEL
LIN {X 0,Y 551.857,Z 338.64,A -85,B 0,C 180,E1 -3181.228,E2 -3181.228} C_VEL
LIN {X 0,Y 551.787,Z 344.437,A -85,B 0,C 180,E1 -3182.341,E2 -3182.341} C_VEL
LIN {X 0,Y 551.746,Z 349.645,A -85,B 0,C 180,E1 -3183.649,E2 -3183.649} C_VEL
LIN {X 0,Y 551.676,Z 353.464,A -85,B 0,C 180,E1 -3184.979,E2 -3184.979} C_VEL
LIN {X 0,Y 551.638,Z 355.231,A -85,B 0,C 180,E1 -3185.878,E2 -3185.878} C_VEL
LIN {X 0,Y 551.645,Z 356.4,A -85,B 0,C 180,E1 -3186.783,E2 -3186.783} C_VEL
LIN {X 0,Y 551.629,Z 356.958,A -85,B 0,C 180,E1 -3187.824,E2 -3187.824} C_VEL
LIN {X 0,Y 551.639,Z 356.637,A -85,B 0,C 180,E1 -3189,E2 -3189} C_VEL
LIN {X 0,Y 551.649,Z 355.328,A -85,B 0,C 180,E1 -3190.147,E2 -3190.147} C_VEL
LIN {X 0,Y 551.719,Z 352.55,A -85,B 0,C 180,E1 -3191.483,E2 -3191.483} C_VEL
LIN {X 0,Y 551.749,Z 349.575,A -85,B 0,C 180,E1 -3192.462,E2 -3192.462} C_VEL
LIN {X 0,Y 551.767,Z 344.622,A -85,B 0,C 180,E1 -3193.71,E2 -3193.71} C_VEL
LIN {X 0,Y 551.87,Z 337.967,A -85,B 0,C 180,E1 -3194.974,E2 -3194.974} C_VEL
LIN {X 0,Y 551.981,Z 330.758,A -85,B 0,C 180,E1 -3196.061,E2 -3196.061} C_VEL
LIN {X 0,Y 552.121,Z 322.446,A -85,B 0,C 180,E1 -3197.079,E2 -3197.079} C_VEL
LIN {X 0,Y 552.278,Z 313.673,A -85,B 0,C 180,E1 -3197.958,E2 -3197.958} C_VEL
LIN {X 0,Y 552.45,Z 303.506,A -85,B 0,C 180,E1 -3198.787,E2 -3198.787} C_VEL
LIN {X 0,Y 552.604,Z 292.593,A -85,B 0,C 180,E1 -3199.503,E2 -3199.503} C_VEL
LIN {X 0,Y 552.866,Z 280.502,A -85,B 0,C 180,E1 -3200.122,E2 -3200.122} C_VEL
LIN {X 0,Y 552.937,Z 267.602,A -85,B 0,C 180,E1 -3200.607,E2 -3200.607} C_VEL
LIN {X 0,Y 553.071,Z 254.517,A -85,B 0,C 180,E1 -3200.937,E2 -3200.937} C_VEL
LIN {X 0,Y 553.265,Z 202.968,A -85,B 0,C 180,E1 -3201.633,E2 -3201.633} C_VEL
LIN {X 0,Y 553.392,Z 153.79,A -85,B 0,C 180,E1 -3202.274,E2 -3202.274} C_VEL
LIN {X 0,Y 552.235,Z 147.174,A -85,B 0,C 180,E1 -3202.406,E2 -3202.406} C_VEL
LIN {X 0,Y 552.373,Z 131.901,A -85,B 0,C 180,E1 -3205.272,E2 -3205.272} C_VEL
LIN {X 0,Y 552.188,Z 124.704,A -85,B 0,C 180,E1 -3206.656,E2 -3206.656} C_VEL
LIN {X 0,Y 552.115,Z 124.709,A -85,B 0,C 180,E1 -3209.951,E2 -3209.951} C_VEL
LIN {X 0,Y 552.14,Z 124.71,A -85,B 0,C 180,E1 -3213.001,E2 -3213.001} C_VEL
LIN {X 0,Y 552.087,Z 124.711,A -85,B 0,C 180,E1 -3215.962,E2 -3215.962} C_VEL
LIN {X 0,Y 552.12,Z 124.714,A -85,B 0,C 180,E1 -3219.12,E2 -3219.12} C_VEL
LIN {X 0,Y 552.091,Z 124.712,A -85,B 0,C 180,E1 -3221.444,E2 -3221.444} C_VEL
LIN {X 0,Y 552.106,Z 124.708,A -85,B 0,C 180,E1 -3223.737,E2 -3223.737} C_VEL
LIN {X 0,Y 552.121,Z 124.707,A -85,B 0,C 180,E1 -3226.005,E2 -3226.005} C_VEL
LIN {X 0,Y 552.163,Z 124.704,A -85,B 0,C 180,E1 -3228.994,E2 -3228.994} C_VEL
LIN {X 0,Y 552.148,Z 124.705,A -85,B 0,C 180,E1 -3231.952,E2 -3231.952} C_VEL
LIN {X 0,Y 552.213,Z 124.697,A -85,B 0,C 180,E1 -3234.889,E2 -3234.889} C_VEL
LIN {X 0,Y 552.223,Z 124.696,A -85,B 0,C 180,E1 -3237.812,E2 -3237.812} C_VEL
LIN {X 0,Y 552.226,Z 124.696,A -85,B 0,C 180,E1 -3240,E2 -3240} C_VEL
LIN {X 0,Y 552.18,Z 124.697,A -85,B 0,C 180,E1 -3242.919,E2 -3242.919} C_VEL
LIN {X 0,Y 552.176,Z 124.705,A -85,B 0,C 180,E1 -3245.845,E2 -3245.845} C_VEL
LIN {X 0,Y 552.126,Z 124.705,A -85,B 0,C 180,E1 -3248.787,E2 -3248.787} C_VEL
LIN {X 0,Y 552.101,Z 124.714,A -85,B 0,C 180,E1 -3251.752,E2 -3251.752} C_VEL
LIN {X 0,Y 552.087,Z 124.708,A -85,B 0,C 180,E1 -3254.75,E2 -3254.75} C_VEL
LIN {X 0,Y 552.068,Z 124.718,A -85,B 0,C 180,E1 -3257.79,E2 -3257.79} C_VEL
LIN {X 0,Y 552.05,Z 124.716,A -85,B 0,C 180,E1 -3260.105,E2 -3260.105} C_VEL
LIN {X 0,Y 552.04,Z 124.715,A -85,B 0,C 180,E1 -3262.454,E2 -3262.454} C_VEL
LIN {X 0,Y 552.068,Z 124.721,A -85,B 0,C 180,E1 -3265.33,E2 -3265.33} C_VEL
LIN {X 0,Y 552.052,Z 124.713,A -85,B 0,C 180,E1 -3268.102,E2 -3268.102} C_VEL
LIN {X 0,Y 552.073,Z 124.714,A -85,B 0,C 180,E1 -3270.611,E2 -3270.611} C_VEL
LIN {X 0,Y 552.108,Z 124.714,A -85,B 0,C 180,E1 -3273.187,E2 -3273.187} C_VEL
LIN {X 0,Y 552.075,Z 124.711,A -85,B 0,C 180,E1 -3275.845,E2 -3275.845} C_VEL
LIN {X 0,Y 552.117,Z 124.711,A -85,B 0,C 180,E1 -3278.589,E2 -3278.589} C_VEL
LIN {X 0,Y 552.079,Z 124.712,A -85,B 0,C 180,E1 -3281.45,E2 -3281.45} C_VEL
LIN {X 0,Y 552.08,Z 124.719,A -85,B 0,C 180,E1 -3284.529,E2 -3284.529} C_VEL
LIN {X 0,Y 552.112,Z 124.708,A -85,B 0,C 180,E1 -3287.587,E2 -3287.587} C_VEL
LIN {X 0,Y 552.131,Z 124.713,A -85,B 0,C 180,E1 -3290.472,E2 -3290.472} C_VEL
LIN {X 0,Y 552.104,Z 124.708,A -85,B 0,C 180,E1 -3293.318,E2 -3293.318} C_VEL
LIN {X 0,Y 552.13,Z 124.71,A -85,B 0,C 180,E1 -3295.939,E2 -3295.939} C_VEL
LIN {X 0,Y 552.125,Z 124.71,A -85,B 0,C 180,E1 -3298.54,E2 -3298.54} C_VEL
LIN {X 0,Y 552.107,Z 124.71,A -85,B 0,C 180,E1 -3301.442,E2 -3301.442} C_VEL
LIN {X 0,Y 552.127,Z 124.711,A -85,B 0,C 180,E1 -3304.355,E2 -3304.355} C_VEL
LIN {X 0,Y 552.166,Z 124.749,A -85,B 0,C 180,E1 -3305.79,E2 -3305.79} C_VEL
LIN {X 0,Y 553.11,Z 131.497,A -85,B 0,C 180,E1 -3306.802,E2 -3306.802} C_VEL
LIN {X 0,Y 552.858,Z 153.344,A -85,B 0,C 180,E1 -3309.926,E2 -3309.926} C_VEL
LIN {X 0,Y 552.605,Z 173.436,A -85,B 0,C 180,E1 -3312.758,E2 -3312.758} C_VEL
LIN {X 0,Y 552.367,Z 193.998,A -85,B 0,C 180,E1 -3315.625,E2 -3315.625} C_VEL
LIN {X 0,Y 553.381,Z 202.031,A -85,B 0,C 180,E1 -3315.761,E2 -3315.761} C_VEL
LIN {X 0,Y 553.139,Z 302.409,A -85,B 0,C 180,E1 -3317.082,E2 -3317.082} C_VEL
LIN {X 0,Y 552.957,Z 315.783,A -85,B 0,C 180,E1 -3317.405,E2 -3317.405} C_VEL
LIN {X 0,Y 552.802,Z 329.145,A -85,B 0,C 180,E1 -3317.891,E2 -3317.891} C_VEL
LIN {X 0,Y 552.651,Z 340.765,A -85,B 0,C 180,E1 -3318.469,E2 -3318.469} C_VEL
LIN {X 0,Y 552.439,Z 352.004,A -85,B 0,C 180,E1 -3319.184,E2 -3319.184} C_VEL
LIN {X 0,Y 552.274,Z 362.493,A -85,B 0,C 180,E1 -3320.015,E2 -3320.015} C_VEL
LIN {X 0,Y 552.132,Z 371.068,A -85,B 0,C 180,E1 -3320.844,E2 -3320.844} C_VEL
LIN {X 0,Y 552.014,Z 378.957,A -85,B 0,C 180,E1 -3321.765,E2 -3321.765} C_VEL
LIN {X 0,Y 551.89,Z 386.618,A -85,B 0,C 180,E1 -3322.867,E2 -3322.867} C_VEL
LIN {X 0,Y 551.868,Z 393.677,A -85,B 0,C 180,E1 -3324.152,E2 -3324.152} C_VEL
LIN {X 0,Y 551.725,Z 398.371,A -85,B 0,C 180,E1 -3325.25,E2 -3325.25} C_VEL
LIN {X 0,Y 551.751,Z 401.957,A -85,B 0,C 180,E1 -3326.348,E2 -3326.348} C_VEL
LIN {X 0,Y 551.724,Z 403.806,A -85,B 0,C 180,E1 -3327.079,E2 -3327.079} C_VEL
LIN {X 0,Y 551.645,Z 406.181,A -85,B 0,C 180,E1 -3328.54,E2 -3328.54} C_VEL
LIN {X 0,Y 551.64,Z 407,A -85,B 0,C 180,E1 -3330,E2 -3330} C_VEL
LIN {X 0,Y 551.645,Z 406.184,A -85,B 0,C 180,E1 -3331.46,E2 -3331.46} C_VEL
LIN {X 0,Y 551.723,Z 403.811,A -85,B 0,C 180,E1 -3332.92,E2 -3332.92} C_VEL
LIN {X 0,Y 551.764,Z 400.896,A -85,B 0,C 180,E1 -3334.017,E2 -3334.017} C_VEL
LIN {X 0,Y 551.723,Z 396.95,A -85,B 0,C 180,E1 -3335.115,E2 -3335.115} C_VEL
LIN {X 0,Y 551.823,Z 391.198,A -85,B 0,C 180,E1 -3336.339,E2 -3336.339} C_VEL
LIN {X 0,Y 551.926,Z 384.238,A -85,B 0,C 180,E1 -3337.499,E2 -3337.499} C_VEL
LIN {X 0,Y 552.082,Z 375.99,A -85,B 0,C 180,E1 -3338.602,E2 -3338.602} C_VEL
LIN {X 0,Y 552.2,Z 367.48,A -85,B 0,C 180,E1 -3339.523,E2 -3339.523} C_VEL
LIN {X 0,Y 552.412,Z 356.961,A -85,B 0,C 180,E1 -3340.445,E2 -3340.445} C_VEL
LIN {X 0,Y 552.555,Z 346.087,A -85,B 0,C 180,E1 -3341.214,E2 -3341.214} C_VEL
LIN {X 0,Y 552.752,Z 335.146,A -85,B 0,C 180,E1 -3341.83,E2 -3341.83} C_VEL
LIN {X 0,Y 552.9,Z 323.436,A -85,B 0,C 180,E1 -3342.339,E2 -3342.339} C_VEL
LIN {X 0,Y 553.053,Z 310.861,A -85,B 0,C 180,E1 -3342.732,E2 -3342.732} C_VEL
LIN {X 0,Y 553.16,Z 298.106,A -85,B 0,C 180,E1 -3342.986,E2 -3342.986} C_VEL
LIN {X 0,Y 553.243,Z 200.11,A -85,B 0,C 180,E1 -3344.268,E2 -3344.268} C_VEL
LIN {X 0,Y 552.36,Z 193.989,A -85,B 0,C 180,E1 -3344.392,E2 -3344.392} C_VEL
LIN {X 0,Y 552.602,Z 173.676,A -85,B 0,C 180,E1 -3347.239,E2 -3347.239} C_VEL
LIN {X 0,Y 552.858,Z 153.687,A -85,B 0,C 180,E1 -3350.073,E2 -3350.073} C_VEL
LIN {X 0,Y 553.225,Z 133.403,A -85,B 0,C 180,E1 -3352.994,E2 -3352.994} C_VEL
LIN {X 0,Y 552.869,Z 128.301,A -85,B 0,C 180,E1 -3353.757,E2 -3353.757} C_VEL
LIN {X 0,Y 552.12,Z 124.715,A -85,B 0,C 180,E1 -3354.337,E2 -3354.337} C_VEL
LIN {X 0,Y 552.135,Z 124.706,A -85,B 0,C 180,E1 -3356.998,E2 -3356.998} C_VEL
LIN {X 0,Y 552.117,Z 124.715,A -85,B 0,C 180,E1 -3360.05,E2 -3360.05} C_VEL
LIN {X 0,Y 552.115,Z 124.706,A -85,B 0,C 180,E1 -3362.846,E2 -3362.846} C_VEL
LIN {X 0,Y 552.077,Z 124.713,A -85,B 0,C 180,E1 -3365.439,E2 -3365.439} C_VEL
LIN {X 0,Y 552.098,Z 124.717,A -85,B 0,C 180,E1 -3367.885,E2 -3367.885} C_VEL
LIN {X 0,Y 552.11,Z 124.708,A -85,B 0,C 180,E1 -3370.481,E2 -3370.481} C_VEL
LIN {X 0,Y 552.107,Z 124.711,A -85,B 0,C 180,E1 -3373.423,E2 -3373.423} C_VEL
LIN {X 0,Y 552.107,Z 124.707,A -85,B 0,C 180,E1 -3376.576,E2 -3376.576} C_VEL
LIN {X 0,Y 552.11,Z 124.714,A -85,B 0,C 180,E1 -3379.519,E2 -3379.519} C_VEL
LIN {X 0,Y 552.092,Z 124.709,A -85,B 0,C 180,E1 -3382.336,E2 -3382.336} C_VEL
LIN {X 0,Y 552.082,Z 124.712,A -85,B 0,C 180,E1 -3385.05,E2 -3385.05} C_VEL
LIN {X 0,Y 552.114,Z 124.713,A -85,B 0,C 180,E1 -3387.681,E2 -3387.681} C_VEL
LIN {X 0,Y 552.108,Z 124.707,A -85,B 0,C 180,E1 -3390.234,E2 -3390.234} C_VEL
LIN {X 0,Y 552.138,Z 124.706,A -85,B 0,C 180,E1 -3393,E2 -3393} C_VEL
LIN {X 0,Y 552.113,Z 124.713,A -85,B 0,C 180,E1 -3395.161,E2 -3395.161} C_VEL
LIN {X 0,Y 552.125,Z 124.704,A -85,B 0,C 180,E1 -3398.337,E2 -3398.337} C_VEL
LIN {X 0,Y 552.15,Z 124.703,A -85,B 0,C 180,E1 -3400.674,E2 -3400.674} C_VEL
LIN {X 0,Y 552.113,Z 124.708,A -85,B 0,C 180,E1 -3403.737,E2 -3403.737} C_VEL
LIN {X 0,Y 552.135,Z 124.703,A -85,B 0,C 180,E1 -3406.004,E2 -3406.004} C_VEL
LIN {X 0,Y 552.162,Z 124.708,A -85,B 0,C 180,E1 -3408.993,E2 -3408.993} C_VEL
LIN {X 0,Y 552.157,Z 124.7,A -85,B 0,C 180,E1 -3411.951,E2 -3411.951} C_VEL
LIN {X 0,Y 552.227,Z 124.701,A -85,B 0,C 180,E1 -3414.889,E2 -3414.889} C_VEL
LIN {X 0,Y 552.225,Z 124.692,A -85,B 0,C 180,E1 -3417.812,E2 -3417.812} C_VEL
LIN {X 0,Y 552.243,Z 124.698,A -85,B 0,C 180,E1 -3420.729,E2 -3420.729} C_VEL
LIN {X 0,Y 552.203,Z 124.702,A -85,B 0,C 180,E1 -3422.918,E2 -3422.918} C_VEL
LIN {X 0,Y 552.201,Z 124.695,A -85,B 0,C 180,E1 -3425.843,E2 -3425.843} C_VEL
LIN {X 0,Y 552.161,Z 124.708,A -85,B 0,C 180,E1 -3428.785,E2 -3428.785} C_VEL
LIN {X 0,Y 552.16,Z 124.7,A -85,B 0,C 180,E1 -3431.75,E2 -3431.75} C_VEL
LIN {X 0,Y 552.134,Z 124.71,A -85,B 0,C 180,E1 -3434.748,E2 -3434.748} C_VEL
LIN {X 0,Y 552.108,Z 124.707,A -85,B 0,C 180,E1 -3437.788,E2 -3437.788} C_VEL
LIN {X 0,Y 552.128,Z 124.708,A -85,B 0,C 180,E1 -3440.101,E2 -3440.101} C_VEL
LIN {X 0,Y 552.09,Z 124.717,A -85,B 0,C 180,E1 -3442.451,E2 -3442.451} C_VEL
LIN {X 0,Y 552.154,Z 124.701,A -85,B 0,C 180,E1 -3445.351,E2 -3445.351} C_VEL
LIN {X 0,Y 552.123,Z 124.711,A -85,B 0,C 180,E1 -3448.097,E2 -3448.097} C_VEL
LIN {X 0,Y 552.104,Z 124.711,A -85,B 0,C 180,E1 -3450.615,E2 -3450.615} C_VEL
LIN {X 0,Y 552.119,Z 124.705,A -85,B 0,C 180,E1 -3453.185,E2 -3453.185} C_VEL
LIN {X 0,Y 552.109,Z 124.711,A -85,B 0,C 180,E1 -3453.795,E2 -3453.795} C_VEL
LIN {X 0,Y 551.472,Z 124.795,A -85,B 0,C 180,E1 -3454.403,E2 -3454.403} C_VEL
LIN {X 0,Y 548.651,Z 125.146,A -85,B 0,C 180,E1 -3455.392,E2 -3455.392} C_VEL
LIN {X 0,Y 546.232,Z 125.447,A -85,B 0,C 180,E1 -3456.187,E2 -3456.187} C_VEL
LIN {X 0,Y 545.163,Z 125.573,A -85,B 0,C 180,E1 -3456.801,E2 -3456.801} C_VEL
LIN {X 0,Y 545.061,Z 125.584,A -85,B 0,C 180,E1 -3457.009,E2 -3457.009} C_VEL
LIN {X 0,Y 545.089,Z 125.589,A -85,B 0,C 180,E1 -3460.14,E2 -3460.14} C_VEL
LIN {X 0,Y 545.082,Z 125.582,A -85,B 0,C 180,E1 -3463.106,E2 -3463.106} C_VEL
LIN {X 0,Y 545.06,Z 125.589,A -85,B 0,C 180,E1 -3466.224,E2 -3466.224} C_VEL
LIN {X 0,Y 545.097,Z 125.58,A -85,B 0,C 180,E1 -3468.887,E2 -3468.887} C_VEL
LIN {X 0,Y 545.051,Z 125.595,A -85,B 0,C 180,E1 -3471.763,E2 -3471.763} C_VEL
LIN {X 0,Y 545.048,Z 125.586,A -85,B 0,C 180,E1 -3474.533,E2 -3474.533} C_VEL
LIN {X 0,Y 545.078,Z 125.585,A -85,B 0,C 180,E1 -3477.213,E2 -3477.213} C_VEL
LIN {X 0,Y 545.062,Z 125.591,A -85,B 0,C 180,E1 -3479.811,E2 -3479.811} C_VEL
LIN {X 0,Y 545.089,Z 125.581,A -85,B 0,C 180,E1 -3482.345,E2 -3482.345} C_VEL
LIN {X 0,Y 545.113,Z 125.579,A -85,B 0,C 180,E1 -3484.821,E2 -3484.821} C_VEL
LIN {X 0,Y 545.04,Z 125.593,A -85,B 0,C 180,E1 -3487.243,E2 -3487.243} C_VEL
LIN {X 0,Y 545.117,Z 125.577,A -85,B 0,C 180,E1 -3490.415,E2 -3490.415} C_VEL
LIN {X 0,Y 545.07,Z 125.59,A -85,B 0,C 180,E1 -3493.522,E2 -3493.522} C_VEL
LIN {X 0,Y 545.091,Z 125.583,A -85,B 0,C 180,E1 -3495.82,E2 -3495.82} C_VEL
LIN {X 0,Y 545.115,Z 125.581,A -85,B 0,C 180,E1 -3498.85,E2 -3498.85} C_VEL
LIN {X 0,Y 545.127,Z 125.577,A -85,B 0,C 180,E1 -3501.847,E2 -3501.847} C_VEL
LIN {X 0,Y 545.204,Z 125.572,A -85,B 0,C 180,E1 -3504.823,E2 -3504.823} C_VEL
LIN {X 0,Y 545.196,Z 125.568,A -85,B 0,C 180,E1 -3507.784,E2 -3507.784} C_VEL
LIN {X 0,Y 545.21,Z 125.571,A -85,B 0,C 180,E1 -3510.739,E2 -3510.739} C_VEL
LIN {X 0,Y 545.169,Z 125.581,A -85,B 0,C 180,E1 -3512.956,E2 -3512.956} C_VEL
LIN {X 0,Y 545.178,Z 125.57,A -85,B 0,C 180,E1 -3515.92,E2 -3515.92} C_VEL
LIN {X 0,Y 545.119,Z 125.586,A -85,B 0,C 180,E1 -3518.9,E2 -3518.9} C_VEL
LIN {X 0,Y 545.133,Z 125.576,A -85,B 0,C 180,E1 -3521.905,E2 -3521.905} C_VEL
LIN {X 0,Y 545.084,Z 125.589,A -85,B 0,C 180,E1 -3524.944,E2 -3524.944} C_VEL
LIN {X 0,Y 545.079,Z 125.586,A -85,B 0,C 180,E1 -3528.026,E2 -3528.026} C_VEL
LIN {X 0,Y 545.168,Z 125.729,A -85,B 0,C 180,E1 -3529.339,E2 -3529.339} C_VEL
LIN {X 0,Y 545.386,Z 132.001,A -85,B 0,C 180,E1 -3530.558,E2 -3530.558} C_VEL
LIN {X 0,Y 545.224,Z 146.596,A -85,B 0,C 180,E1 -3533.352,E2 -3533.352} C_VEL
LIN {X 0,Y 545.206,Z 147.409,A -85,B 0,C 180,E1 -3533.504,E2 -3533.504} C_VEL
LIN {X 0,Y 546.555,Z 155.603,A -85,B 0,C 180,E1 -3533.655,E2 -3533.655} C_VEL
LIN {X 0,Y 546.158,Z 254.103,A -85,B 0,C 180,E1 -3534.976,E2 -3534.976} C_VEL
LIN {X 0,Y 546.029,Z 267.521,A -85,B 0,C 180,E1 -3535.314,E2 -3535.314} C_VEL
LIN {X 0,Y 545.879,Z 279.983,A -85,B 0,C 180,E1 -3535.779,E2 -3535.779} C_VEL
LIN {X 0,Y 545.724,Z 291.796,A -85,B 0,C 180,E1 -3536.379,E2 -3536.379} C_VEL
LIN {X 0,Y 545.459,Z 303.783,A -85,B 0,C 180,E1 -3537.166,E2 -3537.166} C_VEL
LIN {X 0,Y 545.289,Z 313.43,A -85,B 0,C 180,E1 -3537.958,E2 -3537.958} C_VEL
LIN {X 0,Y 545.115,Z 322.159,A -85,B 0,C 180,E1 -3538.831,E2 -3538.831} C_VEL
LIN {X 0,Y 544.959,Z 329.919,A -85,B 0,C 180,E1 -3539.77,E2 -3539.77} C_VEL
LIN {X 0,Y 544.85,Z 337.191,A -85,B 0,C 180,E1 -3540.846,E2 -3540.846} C_VEL
LIN {X 0,Y 544.76,Z 344.197,A -85,B 0,C 180,E1 -3542.153,E2 -3542.153} C_VEL
LIN {X 0,Y 544.661,Z 349.031,A -85,B 0,C 180,E1 -3543.319,E2 -3543.319} C_VEL
LIN {X 0,Y 544.608,Z 352.943,A -85,B 0,C 180,E1 -3544.598,E2 -3544.598} C_VEL
LIN {X 0,Y 544.564,Z 355.118,A -85,B 0,C 180,E1 -3545.605,E2 -3545.605} C_VEL
LIN {X 0,Y 544.561,Z 356.761,A -85,B 0,C 180,E1 -3546.856,E2 -3546.856} C_VEL
LIN {X 0,Y 544.525,Z 357.226,A -85,B 0,C 180,E1 -3548.282,E2 -3548.282} C_VEL
LIN {X 0,Y 544.545,Z 356.747,A -85,B 0,C 180,E1 -3549.253,E2 -3549.253} C_VEL
LIN {X 0,Y 544.571,Z 355.256,A -85,B 0,C 180,E1 -3550.411,E2 -3550.411} C_VEL
LIN {X 0,Y 544.643,Z 352.816,A -85,B 0,C 180,E1 -3551.547,E2 -3551.547} C_VEL
LIN {X 0,Y 544.668,Z 349.459,A -85,B 0,C 180,E1 -3552.652,E2 -3552.652} C_VEL
LIN {X 0,Y 544.707,Z 344.292,A -85,B 0,C 180,E1 -3553.923,E2 -3553.923} C_VEL
LIN {X 0,Y 544.821,Z 337.516,A -85,B 0,C 180,E1 -3555.193,E2 -3555.193} C_VEL
LIN {X 0,Y 544.939,Z 330.536,A -85,B 0,C 180,E1 -3556.239,E2 -3556.239} C_VEL
LIN {X 0,Y 545.134,Z 321.852,A -85,B 0,C 180,E1 -3557.296,E2 -3557.296} C_VEL
LIN {X 0,Y 545.299,Z 312.663,A -85,B 0,C 180,E1 -3558.203,E2 -3558.203} C_VEL
LIN {X 0,Y 545.526,Z 301.713,A -85,B 0,C 180,E1 -3559.077,E2 -3559.077} C_VEL
LIN {X 0,Y 545.69,Z 292.142,A -85,B 0,C 180,E1 -3559.694,E2 -3559.694} C_VEL
LIN {X 0,Y 545.938,Z 280.521,A -85,B 0,C 180,E1 -3560.289,E2 -3560.289} C_VEL
LIN {X 0,Y 546.028,Z 267.236,A -85,B 0,C 180,E1 -3560.787,E2 -3560.787} C_VEL
LIN {X 0,Y 546.169,Z 254.258,A -85,B 0,C 180,E1 -3561.111,E2 -3561.111} C_VEL
LIN {X 0,Y 546.58,Z 154.99,A -85,B 0,C 180,E1 -3562.443,E2 -3562.443} C_VEL
LIN {X 0,Y 545.267,Z 147.414,A -85,B 0,C 180,E1 -3562.599,E2 -3562.599} C_VEL
LIN {X 0,Y 545.376,Z 131.619,A -85,B 0,C 180,E1 -3565.563,E2 -3565.563} C_VEL
LIN {X 0,Y 545.152,Z 125.581,A -85,B 0,C 180,E1 -3566.711,E2 -3566.711} C_VEL
LIN {X 0,Y 545.063,Z 125.589,A -85,B 0,C 180,E1 -3569.811,E2 -3569.811} C_VEL
LIN {X 0,Y 545.08,Z 125.584,A -85,B 0,C 180,E1 -3572.344,E2 -3572.344} C_VEL
LIN {X 0,Y 545.079,Z 125.589,A -85,B 0,C 180,E1 -3574.819,E2 -3574.819} C_VEL
LIN {X 0,Y 545.035,Z 125.597,A -85,B 0,C 180,E1 -3577.243,E2 -3577.243} C_VEL
LIN {X 0,Y 545.12,Z 125.581,A -85,B 0,C 180,E1 -3580.415,E2 -3580.415} C_VEL
LIN {X 0,Y 545.057,Z 125.587,A -85,B 0,C 180,E1 -3583.521,E2 -3583.521} C_VEL
LIN {X 0,Y 545.085,Z 125.583,A -85,B 0,C 180,E1 -3585.82,E2 -3585.82} C_VEL
LIN {X 0,Y 545.12,Z 125.584,A -85,B 0,C 180,E1 -3588.85,E2 -3588.85} C_VEL
LIN {X 0,Y 545.096,Z 125.583,A -85,B 0,C 180,E1 -3591.847,E2 -3591.847} C_VEL
LIN {X 0,Y 545.171,Z 125.575,A -85,B 0,C 180,E1 -3594.823,E2 -3594.823} C_VEL
LIN {X 0,Y 545.194,Z 125.571,A -85,B 0,C 180,E1 -3597.784,E2 -3597.784} C_VEL
LIN {X 0,Y 545.195,Z 125.572,A -85,B 0,C 180,E1 -3600,E2 -3600} C_VEL
LIN {X 0,Y 545.148,Z 125.573,A -85,B 0,C 180,E1 -3602.956,E2 -3602.956} C_VEL
LIN {X 0,Y 545.127,Z 125.585,A -85,B 0,C 180,E1 -3605.92,E2 -3605.92} C_VEL
LIN {X 0,Y 545.07,Z 125.584,A -85,B 0,C 180,E1 -3608.901,E2 -3608.901} C_VEL
LIN {X 0,Y 545.066,Z 125.592,A -85,B 0,C 180,E1 -3611.906,E2 -3611.906} C_VEL
LIN {X 0,Y 545.039,Z 125.587,A -85,B 0,C 180,E1 -3614.945,E2 -3614.945} C_VEL
LIN {X 0,Y 545.034,Z 125.591,A -85,B 0,C 180,E1 -3618.028,E2 -3618.028} C_VEL
LIN {X 0,Y 545.005,Z 125.592,A -85,B 0,C 180,E1 -3620.376,E2 -3620.376} C_VEL
LIN {X 0,Y 544.988,Z 125.595,A -85,B 0,C 180,E1 -3622.76,E2 -3622.76} C_VEL
LIN {X 0,Y 545.02,Z 125.597,A -85,B 0,C 180,E1 -3625.491,E2 -3625.491} C_VEL
LIN {X 0,Y 545.002,Z 125.594,A -85,B 0,C 180,E1 -3627.661,E2 -3627.661} C_VEL
LIN {X 0,Y 545.024,Z 125.59,A -85,B 0,C 180,E1 -3630.236,E2 -3630.236} C_VEL
LIN {X 0,Y 545.075,Z 125.592,A -85,B 0,C 180,E1 -3633.061,E2 -3633.061} C_VEL
LIN {X 0,Y 545.025,Z 125.59,A -85,B 0,C 180,E1 -3635.671,E2 -3635.671} C_VEL
LIN {X 0,Y 545.051,Z 125.587,A -85,B 0,C 180,E1 -3638.238,E2 -3638.238} C_VEL
LIN {X 0,Y 545.033,Z 125.592,A -85,B 0,C 180,E1 -3641.12,E2 -3641.12} C_VEL
LIN {X 0,Y 545.036,Z 125.591,A -85,B 0,C 180,E1 -3644.132,E2 -3644.132} C_VEL
LIN {X 0,Y 545.027,Z 125.595,A -85,B 0,C 180,E1 -3646.888,E2 -3646.888} C_VEL
LIN {X 0,Y 545.084,Z 125.583,A -85,B 0,C 180,E1 -3649.527,E2 -3649.527} C_VEL
LIN {X 0,Y 545.05,Z 125.59,A -85,B 0,C 180,E1 -3651.865,E2 -3651.865} C_VEL
LIN {X 0,Y 545.034,Z 125.594,A -85,B 0,C 180,E1 -3654.531,E2 -3654.531} C_VEL
LIN {X 0,Y 545.071,Z 125.586,A -85,B 0,C 180,E1 -3657.211,E2 -3657.211} C_VEL
LIN {X 0,Y 545.066,Z 125.592,A -85,B 0,C 180,E1 -3659.81,E2 -3659.81} C_VEL
LIN {X 0,Y 545.062,Z 125.591,A -85,B 0,C 180,E1 -3662.342,E2 -3662.342} C_VEL
LIN {X 0,Y 545.111,Z 125.583,A -85,B 0,C 180,E1 -3664.82,E2 -3664.82} C_VEL
LIN {X 0,Y 545.121,Z 125.685,A -85,B 0,C 180,E1 -3665.654,E2 -3665.654} C_VEL
LIN {X 0,Y 546.147,Z 132.47,A -85,B 0,C 180,E1 -3666.69,E2 -3666.69} C_VEL
LIN {X 0,Y 545.927,Z 152.971,A -85,B 0,C 180,E1 -3669.66,E2 -3669.66} C_VEL
LIN {X 0,Y 545.579,Z 174.723,A -85,B 0,C 180,E1 -3672.765,E2 -3672.765} C_VEL
LIN {X 0,Y 545.29,Z 193.711,A -85,B 0,C 180,E1 -3675.439,E2 -3675.439} C_VEL
LIN {X 0,Y 546.502,Z 202.756,A -85,B 0,C 180,E1 -3675.594,E2 -3675.594} C_VEL
LIN {X 0,Y 546.185,Z 303.042,A -85,B 0,C 180,E1 -3676.939,E2 -3676.939} C_VEL
LIN {X 0,Y 545.992,Z 316.086,A -85,B 0,C 180,E1 -3677.265,E2 -3677.265} C_VEL
LIN {X 0,Y 545.838,Z 328.716,A -85,B 0,C 180,E1 -3677.734,E2 -3677.734} C_VEL
LIN {X 0,Y 545.638,Z 340.36,A -85,B 0,C 180,E1 -3678.319,E2 -3678.319} C_VEL
LIN {X 0,Y 545.435,Z 351.613,A -85,B 0,C 180,E1 -3679.044,E2 -3679.044} C_VEL
LIN {X 0,Y 545.229,Z 362.112,A -85,B 0,C 180,E1 -3679.884,E2 -3679.884} C_VEL
LIN {X 0,Y 545.088,Z 370.699,A -85,B 0,C 180,E1 -3680.725,E2 -3680.725} C_VEL
LIN {X 0,Y 544.947,Z 378.62,A -85,B 0,C 180,E1 -3681.657,E2 -3681.657} C_VEL
LIN {X 0,Y 544.825,Z 386.356,A -85,B 0,C 180,E1 -3682.774,E2 -3682.774} C_VEL
LIN {X 0,Y 544.777,Z 393.487,A -85,B 0,C 180,E1 -3684.076,E2 -3684.076} C_VEL
LIN {X 0,Y 544.629,Z 398.225,A -85,B 0,C 180,E1 -3685.188,E2 -3685.188} C_VEL
LIN {X 0,Y 544.669,Z 401.851,A -85,B 0,C 180,E1 -3686.3,E2 -3686.3} C_VEL
LIN {X 0,Y 544.651,Z 403.72,A -85,B 0,C 180,E1 -3687.041,E2 -3687.041} C_VEL
LIN {X 0,Y 544.546,Z 406.116,A -85,B 0,C 180,E1 -3688.52,E2 -3688.52} C_VEL
LIN {X 0,Y 544.542,Z 406.727,A -85,B 0,C 180,E1 -3689.26,E2 -3689.26} C_VEL
LIN {X 0,Y 544.541,Z 406.944,A -85,B 0,C 180,E1 -3690,E2 -3690} C_VEL
LIN {X 0,Y 544.542,Z 406.728,A -85,B 0,C 180,E1 -3690.739,E2 -3690.739} C_VEL
LIN {X 0,Y 544.572,Z 405.123,A -85,B 0,C 180,E1 -3692.218,E2 -3692.218} C_VEL
LIN {X 0,Y 544.65,Z 403.727,A -85,B 0,C 180,E1 -3692.958,E2 -3692.958} C_VEL
LIN {X 0,Y 544.684,Z 400.783,A -85,B 0,C 180,E1 -3694.069,E2 -3694.069} C_VEL
LIN {X 0,Y 544.653,Z 396.795,A -85,B 0,C 180,E1 -3695.182,E2 -3695.182} C_VEL
LIN {X 0,Y 544.727,Z 391.398,A -85,B 0,C 180,E1 -3696.347,E2 -3696.347} C_VEL
LIN {X 0,Y 544.836,Z 385.207,A -85,B 0,C 180,E1 -3697.411,E2 -3697.411} C_VEL
LIN {X 0,Y 544.971,Z 377.15,A -85,B 0,C 180,E1 -3698.528,E2 -3698.528} C_VEL
LIN {X 0,Y 545.113,Z 368.94,A -85,B 0,C 180,E1 -3699.461,E2 -3699.461} C_VEL
LIN {X 0,Y 545.349,Z 358.93,A -85,B 0,C 180,E1 -3700.394,E2 -3700.394} C_VEL
LIN {X 0,Y 545.529,Z 348.042,A -85,B 0,C 180,E1 -3701.208,E2 -3701.208} C_VEL
LIN {X 0,Y 545.708,Z 336.542,A -85,B 0,C 180,E1 -3701.891,E2 -3701.891} C_VEL
LIN {X 0,Y 545.922,Z 324.265,A -85,B 0,C 180,E1 -3702.452,E2 -3702.452} C_VEL
LIN {X 0,Y 546.104,Z 312.257,A -85,B 0,C 180,E1 -3702.85,E2 -3702.85} C_VEL
LIN {X 0,Y 546.214,Z 299.098,A -85,B 0,C 180,E1 -3703.131,E2 -3703.131} C_VEL
LIN {X 0,Y 546.346,Z 200.645,A -85,B 0,C 180,E1 -3704.44,E2 -3704.44} C_VEL
LIN {X 0,Y 545.349,Z 193.697,A -85,B 0,C 180,E1 -3704.579,E2 -3704.579} C_VEL
LIN {X 0,Y 545.595,Z 173.341,A -85,B 0,C 180,E1 -3707.475,E2 -3707.475} C_VEL
LIN {X 0,Y 545.928,Z 153.401,A -85,B 0,C 180,E1 -3710.339,E2 -3710.339} C_VEL
LIN {X 0,Y 546.318,Z 133.142,A -85,B 0,C 180,E1 -3713.302,E2 -3713.302} C_VEL
LIN {X 0,Y 545.096,Z 125.588,A -85,B 0,C 180,E1 -3714.481,E2 -3714.481} C_VEL
LIN {X 0,Y 545.081,Z 125.584,A -85,B 0,C 180,E1 -3717.17,E2 -3717.17} C_VEL
LIN {X 0,Y 545.079,Z 125.589,A -85,B 0,C 180,E1 -3720.246,E2 -3720.246} C_VEL
LIN {X 0,Y 545.08,Z 125.582,A -85,B 0,C 180,E1 -3723.062,E2 -3723.062} C_VEL
LIN {X 0,Y 545.034,Z 125.593,A -85,B 0,C 180,E1 -3725.672,E2 -3725.672} C_VEL
LIN {X 0,Y 545.053,Z 125.59,A -85,B 0,C 180,E1 -3728.237,E2 -3728.237} C_VEL
LIN {X 0,Y 545.082,Z 125.583,A -85,B 0,C 180,E1 -3730.472,E2 -3730.472} C_VEL
LIN {X 0,Y 545.079,Z 125.583,A -85,B 0,C 180,E1 -3733.106,E2 -3733.106} C_VEL
LIN {X 0,Y 545.067,Z 125.586,A -85,B 0,C 180,E1 -3736.224,E2 -3736.224} C_VEL
LIN {X 0,Y 545.086,Z 125.582,A -85,B 0,C 180,E1 -3738.885,E2 -3738.885} C_VEL
LIN {X 0,Y 545.052,Z 125.593,A -85,B 0,C 180,E1 -3741.762,E2 -3741.762} C_VEL
LIN {X 0,Y 545.035,Z 125.588,A -85,B 0,C 180,E1 -3744.531,E2 -3744.531} C_VEL
LIN {X 0,Y 545.065,Z 125.589,A -85,B 0,C 180,E1 -3747.211,E2 -3747.211} C_VEL
LIN {X 0,Y 545.06,Z 125.589,A -85,B 0,C 180,E1 -3749.81,E2 -3749.81} C_VEL
LIN {X 0,Y 545.08,Z 125.582,A -85,B 0,C 180,E1 -3752.343,E2 -3752.343} C_VEL
LIN {X 0,Y 545.117,Z 125.58,A -85,B 0,C 180,E1 -3754.82,E2 -3754.82} C_VEL
LIN {X 0,Y 545.038,Z 125.596,A -85,B 0,C 180,E1 -3757.242,E2 -3757.242} C_VEL
LIN {X 0,Y 545.115,Z 125.578,A -85,B 0,C 180,E1 -3760.414,E2 -3760.414} C_VEL
LIN {X 0,Y 545.071,Z 125.588,A -85,B 0,C 180,E1 -3763.521,E2 -3763.521} C_VEL
LIN {X 0,Y 545.094,Z 125.581,A -85,B 0,C 180,E1 -3765.82,E2 -3765.82} C_VEL
LIN {X 0,Y 545.117,Z 125.583,A -85,B 0,C 180,E1 -3768.849,E2 -3768.849} C_VEL
LIN {X 0,Y 545.127,Z 125.576,A -85,B 0,C 180,E1 -3771.847,E2 -3771.847} C_VEL
LIN {X 0,Y 545.203,Z 125.574,A -85,B 0,C 180,E1 -3774.823,E2 -3774.823} C_VEL
LIN {X 0,Y 545.197,Z 125.568,A -85,B 0,C 180,E1 -3777.783,E2 -3777.783} C_VEL
LIN {X 0,Y 545.213,Z 125.574,A -85,B 0,C 180,E1 -3780.738,E2 -3780.738} C_VEL
LIN {X 0,Y 545.17,Z 125.578,A -85,B 0,C 180,E1 -3782.955,E2 -3782.955} C_VEL
LIN {X 0,Y 545.171,Z 125.571,A -85,B 0,C 180,E1 -3785.919,E2 -3785.919} C_VEL
LIN {X 0,Y 545.119,Z 125.583,A -85,B 0,C 180,E1 -3788.9,E2 -3788.9} C_VEL
LIN {X 0,Y 545.133,Z 125.576,A -85,B 0,C 180,E1 -3791.904,E2 -3791.904} C_VEL
LIN {X 0,Y 545.083,Z 125.585,A -85,B 0,C 180,E1 -3794.943,E2 -3794.943} C_VEL
LIN {X 0,Y 545.077,Z 125.585,A -85,B 0,C 180,E1 -3798.025,E2 -3798.025} C_VEL
LIN {X 0,Y 545.093,Z 125.589,A -85,B 0,C 180,E1 -3800.372,E2 -3800.372} C_VEL
LIN {X 0,Y 545.078,Z 125.583,A -85,B 0,C 180,E1 -3803.559,E2 -3803.559} C_VEL
LIN {X 0,Y 545.086,Z 125.586,A -85,B 0,C 180,E1 -3806,E2 -3806} C_VEL
LIN {X 0,Y 545.087,Z 125.584,A -85,B 0,C 180,E1 -3808.748,E2 -3808.748} C_VEL
LIN {X 0,Y 545.074,Z 125.585,A -85,B 0,C 180,E1 -3811.682,E2 -3811.682} C_VEL
LIN {X 0,Y 545.073,Z 125.586,A -85,B 0,C 180,E1 -3814.563,E2 -3814.563} C_VEL
LIN {X 0,Y 545.061,Z 125.584,A -85,B 0,C 180,E1 -3817.009,E2 -3817.009} C_VEL
LIN {X 0,Y 544.356,Z 125.677,A -85,B 0,C 180,E1 -3817.625,E2 -3817.625} C_VEL
LIN {X 0,Y 541.502,Z 126.031,A -85,B 0,C 180,E1 -3818.626,E2 -3818.626} C_VEL
LIN {X 0,Y 539.125,Z 126.327,A -85,B 0,C 180,E1 -3819.432,E2 -3819.432} C_VEL
LIN {X 0,Y 538.119,Z 126.458,A -85,B 0,C 180,E1 -3820.054,E2 -3820.054} C_VEL
LIN {X 0,Y 538.043,Z 126.459,A -85,B 0,C 180,E1 -3820.265,E2 -3820.265} C_VEL
LIN {X 0,Y 538.028,Z 126.46,A -85,B 0,C 180,E1 -3822.988,E2 -3822.988} C_VEL
LIN {X 0,Y 538.025,Z 126.47,A -85,B 0,C 180,E1 -3825.925,E2 -3825.925} C_VEL
LIN {X 0,Y 538.074,Z 126.456,A -85,B 0,C 180,E1 -3829.249,E2 -3829.249} C_VEL
LIN {X 0,Y 537.991,Z 126.469,A -85,B 0,C 180,E1 -3832.123,E2 -3832.123} C_VEL
LIN {X 0,Y 538.007,Z 126.463,A -85,B 0,C 180,E1 -3834.917,E2 -3834.917} C_VEL
LIN {X 0,Y 538.027,Z 126.47,A -85,B 0,C 180,E1 -3837.618,E2 -3837.618} C_VEL
LIN {X 0,Y 538.014,Z 126.464,A -85,B 0,C 180,E1 -3840.239,E2 -3840.239} C_VEL
LIN {X 0,Y 538.062,Z 126.457,A -85,B 0,C 180,E1 -3842.797,E2 -3842.797} C_VEL
LIN {X 0,Y 538.045,Z 126.464,A -85,B 0,C 180,E1 -3845.293,E2 -3845.293} C_VEL
LIN {X 0,Y 538.011,Z 126.464,A -85,B 0,C 180,E1 -3848.042,E2 -3848.042} C_VEL
LIN {X 0,Y 538.035,Z 126.463,A -85,B 0,C 180,E1 -3850.94,E2 -3850.94} C_VEL
LIN {X 0,Y 538.022,Z 126.47,A -85,B 0,C 180,E1 -3853.299,E2 -3853.299} C_VEL
LIN {X 0,Y 538.06,Z 126.461,A -85,B 0,C 180,E1 -3855.631,E2 -3855.631} C_VEL
LIN {X 0,Y 538.074,Z 126.457,A -85,B 0,C 180,E1 -3858.702,E2 -3858.702} C_VEL
LIN {X 0,Y 538.084,Z 126.455,A -85,B 0,C 180,E1 -3861.74,E2 -3861.74} C_VEL
LIN {X 0,Y 538.162,Z 126.448,A -85,B 0,C 180,E1 -3864.755,E2 -3864.755} C_VEL
LIN {X 0,Y 538.168,Z 126.444,A -85,B 0,C 180,E1 -3867.755,E2 -3867.755} C_VEL
LIN {X 0,Y 538.18,Z 126.447,A -85,B 0,C 180,E1 -3870.749,E2 -3870.749} C_VEL
LIN {X 0,Y 538.136,Z 126.456,A -85,B 0,C 180,E1 -3872.995,E2 -3872.995} C_VEL
LIN {X 0,Y 538.132,Z 126.448,A -85,B 0,C 180,E1 -3875.998,E2 -3875.998} C_VEL
LIN {X 0,Y 538.069,Z 126.462,A -85,B 0,C 180,E1 -3879.018,E2 -3879.018} C_VEL
LIN {X 0,Y 538.081,Z 126.455,A -85,B 0,C 180,E1 -3882.063,E2 -3882.063} C_VEL
LIN {X 0,Y 538.043,Z 126.463,A -85,B 0,C 180,E1 -3885.144,E2 -3885.144} C_VEL
LIN {X 0,Y 538.034,Z 126.467,A -85,B 0,C 180,E1 -3888.271,E2 -3888.271} C_VEL
LIN {X 0,Y 538.107,Z 126.556,A -85,B 0,C 180,E1 -3889.231,E2 -3889.231} C_VEL
LIN {X 0,Y 538.408,Z 132.765,A -85,B 0,C 180,E1 -3890.444,E2 -3890.444} C_VEL
LIN {X 0,Y 538.237,Z 147.814,A -85,B 0,C 180,E1 -3893.317,E2 -3893.317} C_VEL
LIN {X 0,Y 539.7,Z 156.573,A -85,B 0,C 180,E1 -3893.478,E2 -3893.478} C_VEL
LIN {X 0,Y 539.251,Z 254.134,A -85,B 0,C 180,E1 -3894.803,E2 -3894.803} C_VEL
LIN {X 0,Y 539.104,Z 267.659,A -85,B 0,C 180,E1 -3895.145,E2 -3895.145} C_VEL
LIN {X 0,Y 538.951,Z 279.872,A -85,B 0,C 180,E1 -3895.604,E2 -3895.604} C_VEL
LIN {X 0,Y 538.799,Z 291.407,A -85,B 0,C 180,E1 -3896.188,E2 -3896.188} C_VEL
LIN {X 0,Y 538.521,Z 303.307,A -85,B 0,C 180,E1 -3896.969,E2 -3896.969} C_VEL
LIN {X 0,Y 538.281,Z 314.13,A -85,B 0,C 180,E1 -3897.864,E2 -3897.864} C_VEL
LIN {X 0,Y 538.066,Z 324.087,A -85,B 0,C 180,E1 -3898.9,E2 -3898.9} C_VEL
LIN {X 0,Y 537.935,Z 332.09,A -85,B 0,C 180,E1 -3899.925,E2 -3899.925} C_VEL
LIN {X 0,Y 537.758,Z 339.425,A -85,B 0,C 180,E1 -3901.08,E2 -3901.08} C_VEL
LIN {X 0,Y 537.653,Z 345.981,A -85,B 0,C 180,E1 -3902.408,E2 -3902.408} C_VEL
LIN {X 0,Y 537.589,Z 350.992,A -85,B 0,C 180,E1 -3903.753,E2 -3903.753} C_VEL
LIN {X 0,Y 537.499,Z 354.571,A -85,B 0,C 180,E1 -3905.122,E2 -3905.122} C_VEL
LIN {X 0,Y 537.476,Z 356.165,A -85,B 0,C 180,E1 -3906.045,E2 -3906.045} C_VEL
LIN {X 0,Y 537.452,Z 357.249,A -85,B 0,C 180,E1 -3907.093,E2 -3907.093} C_VEL
LIN {X 0,Y 537.433,Z 357.543,A -85,B 0,C 180,E1 -3908.315,E2 -3908.315} C_VEL
LIN {X 0,Y 537.466,Z 356.459,A -85,B 0,C 180,E1 -3909.847,E2 -3909.847} C_VEL
LIN {X 0,Y 537.537,Z 353.784,A -85,B 0,C 180,E1 -3911.32,E2 -3911.32} C_VEL
LIN {X 0,Y 537.598,Z 349.385,A -85,B 0,C 180,E1 -3912.828,E2 -3912.828} C_VEL
LIN {X 0,Y 537.64,Z 344.458,A -85,B 0,C 180,E1 -3914.032,E2 -3914.032} C_VEL
LIN {X 0,Y 537.766,Z 337.893,A -85,B 0,C 180,E1 -3915.277,E2 -3915.277} C_VEL
LIN {X 0,Y 537.92,Z 330.487,A -85,B 0,C 180,E1 -3916.397,E2 -3916.397} C_VEL
LIN {X 0,Y 538.133,Z 321.778,A -85,B 0,C 180,E1 -3917.458,E2 -3917.458} C_VEL
LIN {X 0,Y 538.339,Z 312.437,A -85,B 0,C 180,E1 -3918.382,E2 -3918.382} C_VEL
LIN {X 0,Y 538.533,Z 301.367,A -85,B 0,C 180,E1 -3919.269,E2 -3919.269} C_VEL
LIN {X 0,Y 538.816,Z 290.273,A -85,B 0,C 180,E1 -3919.97,E2 -3919.97} C_VEL
LIN {X 0,Y 539.007,Z 278.807,A -85,B 0,C 180,E1 -3920.533,E2 -3920.533} C_VEL
LIN {X 0,Y 539.144,Z 265.57,A -85,B 0,C 180,E1 -3921.012,E2 -3921.012} C_VEL
LIN {X 0,Y 539.269,Z 252.942,A -85,B 0,C 180,E1 -3921.309,E2 -3921.309} C_VEL
LIN {X 0,Y 539.658,Z 155.456,A -85,B 0,C 180,E1 -3922.63,E2 -3922.63} C_VEL
LIN {X 0,Y 538.279,Z 147.674,A -85,B 0,C 180,E1 -3922.792,E2 -3922.792} C_VEL
LIN {X 0,Y 538.392,Z 132.827,A -85,B 0,C 180,E1 -3925.592,E2 -3925.592} C_VEL
LIN {X 0,Y 538.097,Z 126.46,A -85,B 0,C 180,E1 -3926.809,E2 -3926.809} C_VEL
LIN {X 0,Y 538.017,Z 126.464,A -85,B 0,C 180,E1 -3930.239,E2 -3930.239} C_VEL
LIN {X 0,Y 538.057,Z 126.462,A -85,B 0,C 180,E1 -3932.796,E2 -3932.796} C_VEL
LIN {X 0,Y 538.002,Z 126.473,A -85,B 0,C 180,E1 -3935.291,E2 -3935.291} C_VEL
LIN {X 0,Y 538.018,Z 126.464,A -85,B 0,C 180,E1 -3938.043,E2 -3938.043} C_VEL
LIN {X 0,Y 538.084,Z 126.455,A -85,B 0,C 180,E1 -3940.149,E2 -3940.149} C_VEL
LIN {X 0,Y 538.005,Z 126.468,A -85,B 0,C 180,E1 -3943.299,E2 -3943.299} C_VEL
LIN {X 0,Y 538.058,Z 126.459,A -85,B 0,C 180,E1 -3945.631,E2 -3945.631} C_VEL
LIN {X 0,Y 538.081,Z 126.463,A -85,B 0,C 180,E1 -3948.702,E2 -3948.702} C_VEL
LIN {X 0,Y 538.061,Z 126.459,A -85,B 0,C 180,E1 -3951.74,E2 -3951.74} C_VEL
LIN {X 0,Y 538.131,Z 126.453,A -85,B 0,C 180,E1 -3954.755,E2 -3954.755} C_VEL
LIN {X 0,Y 538.166,Z 126.446,A -85,B 0,C 180,E1 -3957.755,E2 -3957.755} C_VEL
LIN {X 0,Y 538.164,Z 126.448,A -85,B 0,C 180,E1 -3960,E2 -3960} C_VEL
LIN {X 0,Y 538.115,Z 126.449,A -85,B 0,C 180,E1 -3962.995,E2 -3962.995} C_VEL
LIN {X 0,Y 538.083,Z 126.462,A -85,B 0,C 180,E1 -3965.998,E2 -3965.998} C_VEL
LIN {X 0,Y 538.028,Z 126.461,A -85,B 0,C 180,E1 -3969.019,E2 -3969.019} C_VEL
LIN {X 0,Y 538.017,Z 126.467,A -85,B 0,C 180,E1 -3972.064,E2 -3972.064} C_VEL
LIN {X 0,Y 537.988,Z 126.466,A -85,B 0,C 180,E1 -3975.146,E2 -3975.146} C_VEL
LIN {X 0,Y 537.984,Z 126.467,A -85,B 0,C 180,E1 -3978.272,E2 -3978.272} C_VEL
LIN {X 0,Y 537.973,Z 126.468,A -85,B 0,C 180,E1 -3980.654,E2 -3980.654} C_VEL
LIN {X 0,Y 537.977,Z 126.472,A -85,B 0,C 180,E1 -3983.074,E2 -3983.074} C_VEL
LIN {X 0,Y 537.982,Z 126.471,A -85,B 0,C 180,E1 -3985.657,E2 -3985.657} C_VEL
LIN {X 0,Y 537.975,Z 126.467,A -85,B 0,C 180,E1 -3988.054,E2 -3988.054} C_VEL
LIN {X 0,Y 537.992,Z 126.468,A -85,B 0,C 180,E1 -3990.629,E2 -3990.629} C_VEL
LIN {X 0,Y 538.025,Z 126.467,A -85,B 0,C 180,E1 -3993.278,E2 -3993.278} C_VEL
LIN {X 0,Y 537.993,Z 126.465,A -85,B 0,C 180,E1 -3996.005,E2 -3996.005} C_VEL
LIN {X 0,Y 538.013,Z 126.47,A -85,B 0,C 180,E1 -3998.831,E2 -3998.831} C_VEL
LIN {X 0,Y 537.993,Z 126.466,A -85,B 0,C 180,E1 -4001.874,E2 -4001.874} C_VEL
LIN {X 0,Y 537.998,Z 126.471,A -85,B 0,C 180,E1 -4004.863,E2 -4004.863} C_VEL
LIN {X 0,Y 537.991,Z 126.468,A -85,B 0,C 180,E1 -4007.211,E2 -4007.211} C_VEL
LIN {X 0,Y 538.014,Z 126.47,A -85,B 0,C 180,E1 -4010.202,E2 -4010.202} C_VEL
LIN {X 0,Y 538.023,Z 126.463,A -85,B 0,C 180,E1 -4013.066,E2 -4013.066} C_VEL
LIN {X 0,Y 538.022,Z 126.466,A -85,B 0,C 180,E1 -4015.826,E2 -4015.826} C_VEL
LIN {X 0,Y 538.013,Z 126.469,A -85,B 0,C 180,E1 -4018.498,E2 -4018.498} C_VEL
LIN {X 0,Y 538.023,Z 126.463,A -85,B 0,C 180,E1 -4021.097,E2 -4021.097} C_VEL
LIN {X 0,Y 538.038,Z 126.467,A -85,B 0,C 180,E1 -4023.633,E2 -4023.633} C_VEL
LIN {X 0,Y 538.066,Z 126.601,A -85,B 0,C 180,E1 -4025.509,E2 -4025.509} C_VEL
LIN {X 0,Y 539.185,Z 133.452,A -85,B 0,C 180,E1 -4026.574,E2 -4026.574} C_VEL
LIN {X 0,Y 538.922,Z 151.23,A -85,B 0,C 180,E1 -4029.184,E2 -4029.184} C_VEL
LIN {X 0,Y 538.601,Z 171.172,A -85,B 0,C 180,E1 -4032.074,E2 -4032.074} C_VEL
LIN {X 0,Y 538.287,Z 190.637,A -85,B 0,C 180,E1 -4034.863,E2 -4034.863} C_VEL
LIN {X 0,Y 538.252,Z 193.239,A -85,B 0,C 180,E1 -4035.234,E2 -4035.234} C_VEL
LIN {X 0,Y 539.636,Z 204.059,A -85,B 0,C 180,E1 -4035.429,E2 -4035.429} C_VEL
LIN {X 0,Y 539.275,Z 302.528,A -85,B 0,C 180,E1 -4036.768,E2 -4036.768} C_VEL
LIN {X 0,Y 539.052,Z 316.39,A -85,B 0,C 180,E1 -4037.122,E2 -4037.122} C_VEL
LIN {X 0,Y 538.858,Z 329.337,A -85,B 0,C 180,E1 -4037.62,E2 -4037.62} C_VEL
LIN {X 0,Y 538.629,Z 342.04,A -85,B 0,C 180,E1 -4038.29,E2 -4038.29} C_VEL
LIN {X 0,Y 538.367,Z 353.801,A -85,B 0,C 180,E1 -4039.088,E2 -4039.088} C_VEL
LIN {X 0,Y 538.161,Z 362.79,A -85,B 0,C 180,E1 -4039.845,E2 -4039.845} C_VEL
LIN {X 0,Y 537.993,Z 372.022,A -85,B 0,C 180,E1 -4040.791,E2 -4040.791} C_VEL
LIN {X 0,Y 537.815,Z 381.013,A -85,B 0,C 180,E1 -4041.924,E2 -4041.924} C_VEL
LIN {X 0,Y 537.68,Z 388.254,A -85,B 0,C 180,E1 -4043.055,E2 -4043.055} C_VEL
LIN {X 0,Y 537.657,Z 394.849,A -85,B 0,C 180,E1 -4044.373,E2 -4044.373} C_VEL
LIN {X 0,Y 537.553,Z 399.207,A -85,B 0,C 180,E1 -4045.5,E2 -4045.5} C_VEL
LIN {X 0,Y 537.591,Z 401.518,A -85,B 0,C 180,E1 -4046.252,E2 -4046.252} C_VEL
LIN {X 0,Y 537.58,Z 403.39,A -85,B 0,C 180,E1 -4047.002,E2 -4047.002} C_VEL
LIN {X 0,Y 537.452,Z 405.79,A -85,B 0,C 180,E1 -4048.501,E2 -4048.501} C_VEL
LIN {X 0,Y 537.449,Z 406.401,A -85,B 0,C 180,E1 -4049.25,E2 -4049.25} C_VEL
LIN {X 0,Y 537.449,Z 406.621,A -85,B 0,C 180,E1 -4050,E2 -4050} C_VEL
LIN {X 0,Y 537.449,Z 406.405,A -85,B 0,C 180,E1 -4050.749,E2 -4050.749} C_VEL
LIN {X 0,Y 537.49,Z 404.801,A -85,B 0,C 180,E1 -4052.248,E2 -4052.248} C_VEL
LIN {X 0,Y 537.58,Z 403.405,A -85,B 0,C 180,E1 -4052.997,E2 -4052.997} C_VEL
LIN {X 0,Y 537.603,Z 400.46,A -85,B 0,C 180,E1 -4054.123,E2 -4054.123} C_VEL
LIN {X 0,Y 537.587,Z 396.469,A -85,B 0,C 180,E1 -4055.25,E2 -4055.25} C_VEL
LIN {X 0,Y 537.652,Z 390.363,A -85,B 0,C 180,E1 -4056.562,E2 -4056.562} C_VEL
LIN {X 0,Y 537.784,Z 383.631,A -85,B 0,C 180,E1 -4057.698,E2 -4057.698} C_VEL
LIN {X 0,Y 537.93,Z 375.313,A -85,B 0,C 180,E1 -4058.83,E2 -4058.83} C_VEL
LIN {X 0,Y 538.089,Z 366.784,A -85,B 0,C 180,E1 -4059.775,E2 -4059.775} C_VEL
LIN {X 0,Y 538.333,Z 356.247,A -85,B 0,C 180,E1 -4060.721,E2 -4060.721} C_VEL
LIN {X 0,Y 538.574,Z 345.024,A -85,B 0,C 180,E1 -4061.531,E2 -4061.531} C_VEL
LIN {X 0,Y 538.808,Z 334.393,A -85,B 0,C 180,E1 -4062.141,E2 -4062.141} C_VEL
LIN {X 0,Y 538.977,Z 322.626,A -85,B 0,C 180,E1 -4062.663,E2 -4062.663} C_VEL
LIN {X 0,Y 539.211,Z 309.986,A -85,B 0,C 180,E1 -4063.065,E2 -4063.065} C_VEL
LIN {X 0,Y 539.343,Z 297.089,A -85,B 0,C 180,E1 -4063.325,E2 -4063.325} C_VEL
LIN {X 0,Y 539.507,Z 201.63,A -85,B 0,C 180,E1 -4064.609,E2 -4064.609} C_VEL
LIN {X 0,Y 538.298,Z 193.444,A -85,B 0,C 180,E1 -4064.766,E2 -4064.766} C_VEL
LIN {X 0,Y 538.585,Z 174.747,A -85,B 0,C 180,E1 -4067.465,E2 -4067.465} C_VEL
LIN {X 0,Y 538.972,Z 154.177,A -85,B 0,C 180,E1 -4070.457,E2 -4070.457} C_VEL
LIN {X 0,Y 539.396,Z 134.23,A -85,B 0,C 180,E1 -4073.415,E2 -4073.415} C_VEL
LIN {X 0,Y 538.052,Z 126.465,A -85,B 0,C 180,E1 -4074.661,E2 -4074.661} C_VEL
LIN {X 0,Y 538.045,Z 126.462,A -85,B 0,C 180,E1 -4077.349,E2 -4077.349} C_VEL
LIN {X 0,Y 538.028,Z 126.465,A -85,B 0,C 180,E1 -4080.443,E2 -4080.443} C_VEL
LIN {X 0,Y 538.047,Z 126.459,A -85,B 0,C 180,E1 -4083.282,E2 -4083.282} C_VEL
LIN {X 0,Y 537.995,Z 126.473,A -85,B 0,C 180,E1 -4086.004,E2 -4086.004} C_VEL
LIN {X 0,Y 538.015,Z 126.462,A -85,B 0,C 180,E1 -4088.83,E2 -4088.83} C_VEL
LIN {X 0,Y 538.031,Z 126.469,A -85,B 0,C 180,E1 -4091.773,E2 -4091.773} C_VEL
LIN {X 0,Y 538.009,Z 126.463,A -85,B 0,C 180,E1 -4094.861,E2 -4094.861} C_VEL
LIN {X 0,Y 538.019,Z 126.464,A -85,B 0,C 180,E1 -4097.214,E2 -4097.214} C_VEL
LIN {X 0,Y 538.023,Z 126.463,A -85,B 0,C 180,E1 -4100.203,E2 -4100.203} C_VEL
LIN {X 0,Y 538.024,Z 126.463,A -85,B 0,C 180,E1 -4103.067,E2 -4103.067} C_VEL
LIN {X 0,Y 538.01,Z 126.468,A -85,B 0,C 180,E1 -4105.826,E2 -4105.826} C_VEL
LIN {X 0,Y 538.008,Z 126.463,A -85,B 0,C 180,E1 -4108.498,E2 -4108.498} C_VEL
LIN {X 0,Y 538.042,Z 126.463,A -85,B 0,C 180,E1 -4111.098,E2 -4111.098} C_VEL
LIN {X 0,Y 538.041,Z 126.464,A -85,B 0,C 180,E1 -4113.633,E2 -4113.633} C_VEL
LIN {X 0,Y 538.006,Z 126.464,A -85,B 0,C 180,E1 -4116.122,E2 -4116.122} C_VEL
LIN {X 0,Y 538.037,Z 126.468,A -85,B 0,C 180,E1 -4119.348,E2 -4119.348} C_VEL
LIN {X 0,Y 538.035,Z 126.46,A -85,B 0,C 180,E1 -4122.467,E2 -4122.467} C_VEL
LIN {X 0,Y 538.063,Z 126.459,A -85,B 0,C 180,E1 -4125.63,E2 -4125.63} C_VEL
LIN {X 0,Y 538.076,Z 126.458,A -85,B 0,C 180,E1 -4128.701,E2 -4128.701} C_VEL
LIN {X 0,Y 538.084,Z 126.454,A -85,B 0,C 180,E1 -4131.739,E2 -4131.739} C_VEL
LIN {X 0,Y 538.161,Z 126.45,A -85,B 0,C 180,E1 -4134.755,E2 -4134.755} C_VEL
LIN {X 0,Y 538.168,Z 126.443,A -85,B 0,C 180,E1 -4137.754,E2 -4137.754} C_VEL
LIN {X 0,Y 538.183,Z 126.45,A -85,B 0,C 180,E1 -4140.748,E2 -4140.748} C_VEL
LIN {X 0,Y 538.136,Z 126.453,A -85,B 0,C 180,E1 -4142.994,E2 -4142.994} C_VEL
LIN {X 0,Y 538.121,Z 126.45,A -85,B 0,C 180,E1 -4145.997,E2 -4145.997} C_VEL
LIN {X 0,Y 538.07,Z 126.459,A -85,B 0,C 180,E1 -4149.017,E2 -4149.017} C_VEL
LIN {X 0,Y 538.081,Z 126.456,A -85,B 0,C 180,E1 -4152.062,E2 -4152.062} C_VEL
LIN {X 0,Y 538.043,Z 126.46,A -85,B 0,C 180,E1 -4155.143,E2 -4155.143} C_VEL
LIN {X 0,Y 538.029,Z 126.467,A -85,B 0,C 180,E1 -4158.27,E2 -4158.27} C_VEL
LIN {X 0,Y 538.037,Z 126.465,A -85,B 0,C 180,E1 -4160.651,E2 -4160.651} C_VEL
LIN {X 0,Y 538.001,Z 126.467,A -85,B 0,C 180,E1 -4163.888,E2 -4163.888} C_VEL
LIN {X 0,Y 538.047,Z 126.467,A -85,B 0,C 180,E1 -4166.366,E2 -4166.366} C_VEL
LIN {X 0,Y 538.028,Z 126.462,A -85,B 0,C 180,E1 -4168.933,E2 -4168.933} C_VEL
LIN {X 0,Y 538.024,Z 126.466,A -85,B 0,C 180,E1 -4171.89,E2 -4171.89} C_VEL
LIN {X 0,Y 538.023,Z 126.464,A -85,B 0,C 180,E1 -4174.62,E2 -4174.62} C_VEL
LIN {X 0,Y 538.004,Z 126.464,A -85,B 0,C 180,E1 -4177.17,E2 -4177.17} C_VEL
LIN {X 0,Y 538.043,Z 126.459,A -85,B 0,C 180,E1 -4180.265,E2 -4180.265} C_VEL
LIN {X 0,Y 537.391,Z 126.541,A -85,B 0,C 180,E1 -4180.89,E2 -4180.89} C_VEL
LIN {X 0,Y 534.532,Z 126.904,A -85,B 0,C 180,E1 -4181.904,E2 -4181.904} C_VEL
LIN {X 0,Y 532.099,Z 127.207,A -85,B 0,C 180,E1 -4182.721,E2 -4182.721} C_VEL
LIN {X 0,Y 531.047,Z 127.334,A -85,B 0,C 180,E1 -4183.352,E2 -4183.352} C_VEL
LIN {X 0,Y 530.959,Z 127.343,A -85,B 0,C 180,E1 -4183.566,E2 -4183.566} C_VEL
LIN {X 0,Y 530.962,Z 127.342,A -85,B 0,C 180,E1 -4186.506,E2 -4186.506} C_VEL
LIN {X 0,Y 531.022,Z 127.339,A -85,B 0,C 180,E1 -4189.571,E2 -4189.571} C_VEL
LIN {X 0,Y 530.965,Z 127.341,A -85,B 0,C 180,E1 -4192.577,E2 -4192.577} C_VEL
LIN {X 0,Y 530.991,Z 127.341,A -85,B 0,C 180,E1 -4195.311,E2 -4195.311} C_VEL
LIN {X 0,Y 530.978,Z 127.342,A -85,B 0,C 180,E1 -4198.033,E2 -4198.033} C_VEL
LIN {X 0,Y 530.985,Z 127.339,A -85,B 0,C 180,E1 -4200.874,E2 -4200.874} C_VEL
LIN {X 0,Y 531.002,Z 127.341,A -85,B 0,C 180,E1 -4203.257,E2 -4203.257} C_VEL
LIN {X 0,Y 530.993,Z 127.34,A -85,B 0,C 180,E1 -4205.958,E2 -4205.958} C_VEL
LIN {X 0,Y 530.997,Z 127.34,A -85,B 0,C 180,E1 -4209.062,E2 -4209.062} C_VEL
LIN {X 0,Y 531.012,Z 127.335,A -85,B 0,C 180,E1 -4212.278,E2 -4212.278} C_VEL
LIN {X 0,Y 531.037,Z 127.339,A -85,B 0,C 180,E1 -4215.437,E2 -4215.437} C_VEL
LIN {X 0,Y 531.033,Z 127.333,A -85,B 0,C 180,E1 -4218.55,E2 -4218.55} C_VEL
LIN {X 0,Y 531.053,Z 127.332,A -85,B 0,C 180,E1 -4221.63,E2 -4221.63} C_VEL
LIN {X 0,Y 531.122,Z 127.324,A -85,B 0,C 180,E1 -4224.686,E2 -4224.686} C_VEL
LIN {X 0,Y 531.139,Z 127.32,A -85,B 0,C 180,E1 -4227.725,E2 -4227.725} C_VEL
LIN {X 0,Y 531.15,Z 127.323,A -85,B 0,C 180,E1 -4230.759,E2 -4230.759} C_VEL
LIN {X 0,Y 531.102,Z 127.331,A -85,B 0,C 180,E1 -4233.035,E2 -4233.035} C_VEL
LIN {X 0,Y 531.09,Z 127.325,A -85,B 0,C 180,E1 -4236.077,E2 -4236.077} C_VEL
LIN {X 0,Y 531.029,Z 127.337,A -85,B 0,C 180,E1 -4239.139,E2 -4239.139} C_VEL
LIN {X 0,Y 531.039,Z 127.333,A -85,B 0,C 180,E1 -4242.225,E2 -4242.225} C_VEL
LIN {X 0,Y 530.994,Z 127.34,A -85,B 0,C 180,E1 -4245.35,E2 -4245.35} C_VEL
LIN {X 0,Y 531,Z 127.346,A -85,B 0,C 180,E1 -4248.521,E2 -4248.521} C_VEL
LIN {X 0,Y 531.053,Z 127.425,A -85,B 0,C 180,E1 -4249.12,E2 -4249.12} C_VEL
LIN {X 0,Y 531.478,Z 132.559,A -85,B 0,C 180,E1 -4250.139,E2 -4250.139} C_VEL
LIN {X 0,Y 531.22,Z 147.859,A -85,B 0,C 180,E1 -4253.101,E2 -4253.101} C_VEL
LIN {X 0,Y 532.816,Z 156.779,A -85,B 0,C 180,E1 -4253.285,E2 -4253.285} C_VEL
LIN {X 0,Y 532.367,Z 254.174,A -85,B 0,C 180,E1 -4254.627,E2 -4254.627} C_VEL
LIN {X 0,Y 532.202,Z 267.056,A -85,B 0,C 180,E1 -4254.949,E2 -4254.949} C_VEL
LIN {X 0,Y 532.037,Z 279.739,A -85,B 0,C 180,E1 -4255.424,E2 -4255.424} C_VEL
LIN {X 0,Y 531.871,Z 291.719,A -85,B 0,C 180,E1 -4256.035,E2 -4256.035} C_VEL
LIN {X 0,Y 531.608,Z 302.078,A -85,B 0,C 180,E1 -4256.711,E2 -4256.711} C_VEL
LIN {X 0,Y 531.352,Z 313.01,A -85,B 0,C 180,E1 -4257.603,E2 -4257.603} C_VEL
LIN {X 0,Y 531.133,Z 321.462,A -85,B 0,C 180,E1 -4258.448,E2 -4258.448} C_VEL
LIN {X 0,Y 530.931,Z 330.462,A -85,B 0,C 180,E1 -4259.544,E2 -4259.544} C_VEL
LIN {X 0,Y 530.749,Z 338.735,A -85,B 0,C 180,E1 -4260.818,E2 -4260.818} C_VEL
LIN {X 0,Y 530.645,Z 345.046,A -85,B 0,C 180,E1 -4262.046,E2 -4262.046} C_VEL
LIN {X 0,Y 530.496,Z 350.426,A -85,B 0,C 180,E1 -4263.424,E2 -4263.424} C_VEL
LIN {X 0,Y 530.421,Z 354.183,A -85,B 0,C 180,E1 -4264.767,E2 -4264.767} C_VEL
LIN {X 0,Y 530.408,Z 356.567,A -85,B 0,C 180,E1 -4266.075,E2 -4266.075} C_VEL
LIN {X 0,Y 530.342,Z 357.821,A -85,B 0,C 180,E1 -4267.56,E2 -4267.56} C_VEL
LIN {X 0,Y 530.351,Z 357.816,A -85,B 0,C 180,E1 -4268.571,E2 -4268.571} C_VEL
LIN {X 0,Y 530.371,Z 356.889,A -85,B 0,C 180,E1 -4269.776,E2 -4269.776} C_VEL
LIN {X 0,Y 530.453,Z 354.996,A -85,B 0,C 180,E1 -4270.958,E2 -4270.958} C_VEL
LIN {X 0,Y 530.5,Z 350.98,A -85,B 0,C 180,E1 -4272.505,E2 -4272.505} C_VEL
LIN {X 0,Y 530.58,Z 347.266,A -85,B 0,C 180,E1 -4273.535,E2 -4273.535} C_VEL
LIN {X 0,Y 530.66,Z 341.417,A -85,B 0,C 180,E1 -4274.795,E2 -4274.795} C_VEL
LIN {X 0,Y 530.866,Z 333.84,A -85,B 0,C 180,E1 -4276.074,E2 -4276.074} C_VEL
LIN {X 0,Y 531.055,Z 325.867,A -85,B 0,C 180,E1 -4277.143,E2 -4277.143} C_VEL
LIN {X 0,Y 531.287,Z 316.003,A -85,B 0,C 180,E1 -4278.213,E2 -4278.213} C_VEL
LIN {X 0,Y 531.516,Z 305.658,A -85,B 0,C 180,E1 -4279.118,E2 -4279.118} C_VEL
LIN {X 0,Y 531.744,Z 294.56,A -85,B 0,C 180,E1 -4279.889,E2 -4279.889} C_VEL
LIN {X 0,Y 532.05,Z 282.549,A -85,B 0,C 180,E1 -4280.54,E2 -4280.54} C_VEL
LIN {X 0,Y 532.192,Z 269.804,A -85,B 0,C 180,E1 -4281.056,E2 -4281.056} C_VEL
LIN {X 0,Y 532.342,Z 256.354,A -85,B 0,C 180,E1 -4281.419,E2 -4281.419} C_VEL
LIN {X 0,Y 532.522,Z 228.518,A -85,B 0,C 180,E1 -4281.829,E2 -4281.829} C_VEL
LIN {X 0,Y 532.773,Z 156.011,A -85,B 0,C 180,E1 -4282.82,E2 -4282.82} C_VEL
LIN {X 0,Y 531.278,Z 147.94,A -85,B 0,C 180,E1 -4282.995,E2 -4282.995} C_VEL
LIN {X 0,Y 531.404,Z 133.088,A -85,B 0,C 180,E1 -4285.801,E2 -4285.801} C_VEL
LIN {X 0,Y 531.054,Z 127.338,A -85,B 0,C 180,E1 -4286.925,E2 -4286.925} C_VEL
LIN {X 0,Y 530.963,Z 127.346,A -85,B 0,C 180,E1 -4289.803,E2 -4289.803} C_VEL
LIN {X 0,Y 531.014,Z 127.337,A -85,B 0,C 180,E1 -4292.468,E2 -4292.468} C_VEL
LIN {X 0,Y 530.971,Z 127.349,A -85,B 0,C 180,E1 -4294.941,E2 -4294.941} C_VEL
LIN {X 0,Y 530.98,Z 127.341,A -85,B 0,C 180,E1 -4297.899,E2 -4297.899} C_VEL
LIN {X 0,Y 530.986,Z 127.344,A -85,B 0,C 180,E1 -4300.677,E2 -4300.677} C_VEL
LIN {X 0,Y 530.967,Z 127.348,A -85,B 0,C 180,E1 -4303.071,E2 -4303.071} C_VEL
LIN {X 0,Y 531.017,Z 127.337,A -85,B 0,C 180,E1 -4305.436,E2 -4305.436} C_VEL
LIN {X 0,Y 531.039,Z 127.341,A -85,B 0,C 180,E1 -4308.55,E2 -4308.55} C_VEL
LIN {X 0,Y 531.037,Z 127.334,A -85,B 0,C 180,E1 -4311.63,E2 -4311.63} C_VEL
LIN {X 0,Y 531.092,Z 127.33,A -85,B 0,C 180,E1 -4314.685,E2 -4314.685} C_VEL
LIN {X 0,Y 531.137,Z 127.322,A -85,B 0,C 180,E1 -4317.725,E2 -4317.725} C_VEL
LIN {X 0,Y 531.132,Z 127.323,A -85,B 0,C 180,E1 -4320,E2 -4320} C_VEL
LIN {X 0,Y 531.137,Z 127.325,A -85,B 0,C 180,E1 -4322.275,E2 -4322.275} C_VEL
LIN {X 0,Y 531.085,Z 127.327,A -85,B 0,C 180,E1 -4325.316,E2 -4325.316} C_VEL
LIN {X 0,Y 530.986,Z 127.341,A -85,B 0,C 180,E1 -4328.372,E2 -4328.372} C_VEL
LIN {X 0,Y 531.016,Z 127.338,A -85,B 0,C 180,E1 -4331.65,E2 -4331.65} C_VEL
LIN {X 0,Y 530.966,Z 127.339,A -85,B 0,C 180,E1 -4334.927,E2 -4334.927} C_VEL
LIN {X 0,Y 530.949,Z 127.349,A -85,B 0,C 180,E1 -4337.725,E2 -4337.725} C_VEL
LIN {X 0,Y 530.932,Z 127.346,A -85,B 0,C 180,E1 -4340.941,E2 -4340.941} C_VEL
LIN {X 0,Y 530.925,Z 127.352,A -85,B 0,C 180,E1 -4343.399,E2 -4343.399} C_VEL
LIN {X 0,Y 530.929,Z 127.347,A -85,B 0,C 180,E1 -4345.902,E2 -4345.902} C_VEL
LIN {X 0,Y 530.934,Z 127.344,A -85,B 0,C 180,E1 -4348.46,E2 -4348.46} C_VEL
LIN {X 0,Y 530.94,Z 127.351,A -85,B 0,C 180,E1 -4351.081,E2 -4351.081} C_VEL
LIN {X 0,Y 530.955,Z 127.343,A -85,B 0,C 180,E1 -4353.775,E2 -4353.775} C_VEL
LIN {X 0,Y 530.955,Z 127.346,A -85,B 0,C 180,E1 -4356.559,E2 -4356.559} C_VEL
LIN {X 0,Y 530.973,Z 127.342,A -85,B 0,C 180,E1 -4359.445,E2 -4359.445} C_VEL
LIN {X 0,Y 530.924,Z 127.352,A -85,B 0,C 180,E1 -4362.463,E2 -4362.463} C_VEL
LIN {X 0,Y 530.971,Z 127.342,A -85,B 0,C 180,E1 -4365.451,E2 -4365.451} C_VEL
LIN {X 0,Y 530.984,Z 127.347,A -85,B 0,C 180,E1 -4368.563,E2 -4368.563} C_VEL
LIN {X 0,Y 530.958,Z 127.343,A -85,B 0,C 180,E1 -4371.529,E2 -4371.529} C_VEL
LIN {X 0,Y 530.955,Z 127.351,A -85,B 0,C 180,E1 -4374.379,E2 -4374.379} C_VEL
LIN {X 0,Y 530.972,Z 127.343,A -85,B 0,C 180,E1 -4377.133,E2 -4377.133} C_VEL
LIN {X 0,Y 530.963,Z 127.348,A -85,B 0,C 180,E1 -4379.802,E2 -4379.802} C_VEL
LIN {X 0,Y 530.98,Z 127.344,A -85,B 0,C 180,E1 -4382.475,E2 -4382.475} C_VEL
LIN {X 0,Y 531.065,Z 127.52,A -85,B 0,C 180,E1 -4385.363,E2 -4385.363} C_VEL
LIN {X 0,Y 532.218,Z 134.446,A -85,B 0,C 180,E1 -4386.455,E2 -4386.455} C_VEL
LIN {X 0,Y 531.989,Z 148.128,A -85,B 0,C 180,E1 -4388.493,E2 -4388.493} C_VEL
LIN {X 0,Y 531.728,Z 161.759,A -85,B 0,C 180,E1 -4390.504,E2 -4390.504} C_VEL
LIN {X 0,Y 531.462,Z 179.433,A -85,B 0,C 180,E1 -4393.086,E2 -4393.086} C_VEL
LIN {X 0,Y 531.254,Z 193.075,A -85,B 0,C 180,E1 -4395.047,E2 -4395.047} C_VEL
LIN {X 0,Y 532.748,Z 204.864,A -85,B 0,C 180,E1 -4395.253,E2 -4395.253} C_VEL
LIN {X 0,Y 532.367,Z 302.014,A -85,B 0,C 180,E1 -4396.594,E2 -4396.594} C_VEL
LIN {X 0,Y 532.104,Z 315.927,A -85,B 0,C 180,E1 -4396.951,E2 -4396.951} C_VEL
LIN {X 0,Y 531.893,Z 328.916,A -85,B 0,C 180,E1 -4397.455,E2 -4397.455} C_VEL
LIN {X 0,Y 531.632,Z 341.636,A -85,B 0,C 180,E1 -4398.134,E2 -4398.134} C_VEL
LIN {X 0,Y 531.373,Z 353.415,A -85,B 0,C 180,E1 -4398.943,E2 -4398.943} C_VEL
LIN {X 0,Y 531.136,Z 362.413,A -85,B 0,C 180,E1 -4399.709,E2 -4399.709} C_VEL
LIN {X 0,Y 530.96,Z 371.656,A -85,B 0,C 180,E1 -4400.668,E2 -4400.668} C_VEL
LIN {X 0,Y 530.752,Z 380.656,A -85,B 0,C 180,E1 -4401.816,E2 -4401.816} C_VEL
LIN {X 0,Y 530.623,Z 387.905,A -85,B 0,C 180,E1 -4402.962,E2 -4402.962} C_VEL
LIN {X 0,Y 530.571,Z 394.507,A -85,B 0,C 180,E1 -4404.298,E2 -4404.298} C_VEL
LIN {X 0,Y 530.451,Z 398.87,A -85,B 0,C 180,E1 -4405.44,E2 -4405.44} C_VEL
LIN {X 0,Y 530.516,Z 401.185,A -85,B 0,C 180,E1 -4406.202,E2 -4406.202} C_VEL
LIN {X 0,Y 530.483,Z 403.06,A -85,B 0,C 180,E1 -4406.962,E2 -4406.962} C_VEL
LIN {X 0,Y 530.413,Z 404.462,A -85,B 0,C 180,E1 -4407.721,E2 -4407.721} C_VEL
LIN {X 0,Y 530.356,Z 406.077,A -85,B 0,C 180,E1 -4409.24,E2 -4409.24} C_VEL
LIN {X 0,Y 530.357,Z 406.298,A -85,B 0,C 180,E1 -4410,E2 -4410} C_VEL
LIN {X 0,Y 530.356,Z 406.082,A -85,B 0,C 180,E1 -4410.759,E2 -4410.759} C_VEL
LIN {X 0,Y 530.412,Z 404.479,A -85,B 0,C 180,E1 -4412.278,E2 -4412.278} C_VEL
LIN {X 0,Y 530.483,Z 403.081,A -85,B 0,C 180,E1 -4413.037,E2 -4413.037} C_VEL
LIN {X 0,Y 530.521,Z 400.136,A -85,B 0,C 180,E1 -4414.178,E2 -4414.178} C_VEL
LIN {X 0,Y 530.522,Z 396.144,A -85,B 0,C 180,E1 -4415.32,E2 -4415.32} C_VEL
LIN {X 0,Y 530.554,Z 390.624,A -85,B 0,C 180,E1 -4416.539,E2 -4416.539} C_VEL
LIN {X 0,Y 530.704,Z 383.296,A -85,B 0,C 180,E1 -4417.801,E2 -4417.801} C_VEL
LIN {X 0,Y 530.879,Z 374.973,A -85,B 0,C 180,E1 -4418.948,E2 -4418.948} C_VEL
LIN {X 0,Y 531.048,Z 366.436,A -85,B 0,C 180,E1 -4419.906,E2 -4419.906} C_VEL
LIN {X 0,Y 531.294,Z 355.89,A -85,B 0,C 180,E1 -4420.865,E2 -4420.865} C_VEL
LIN {X 0,Y 531.575,Z 345.187,A -85,B 0,C 180,E1 -4421.65,E2 -4421.65} C_VEL
LIN {X 0,Y 531.842,Z 334.016,A -85,B 0,C 180,E1 -4422.303,E2 -4422.303} C_VEL
LIN {X 0,Y 532.036,Z 322.222,A -85,B 0,C 180,E1 -4422.831,E2 -4422.831} C_VEL
LIN {X 0,Y 532.258,Z 308.632,A -85,B 0,C 180,E1 -4423.263,E2 -4423.263} C_VEL
LIN {X 0,Y 532.449,Z 296.583,A -85,B 0,C 180,E1 -4423.501,E2 -4423.501} C_VEL
LIN {X 0,Y 532.623,Z 202.372,A -85,B 0,C 180,E1 -4424.788,E2 -4424.788} C_VEL
LIN {X 0,Y 531.249,Z 193.115,A -85,B 0,C 180,E1 -4424.969,E2 -4424.969} C_VEL
LIN {X 0,Y 531.617,Z 173.415,A -85,B 0,C 180,E1 -4427.853,E2 -4427.853} C_VEL
LIN {X 0,Y 531.981,Z 154.093,A -85,B 0,C 180,E1 -4430.708,E2 -4430.708} C_VEL
LIN {X 0,Y 532.457,Z 135.31,A -85,B 0,C 180,E1 -4433.532,E2 -4433.532} C_VEL
LIN {X 0,Y 531.024,Z 127.34,A -85,B 0,C 180,E1 -4434.847,E2 -4434.847} C_VEL
LIN {X 0,Y 531.01,Z 127.34,A -85,B 0,C 180,E1 -4437.595,E2 -4437.595} C_VEL
LIN {X 0,Y 530.975,Z 127.341,A -85,B 0,C 180,E1 -4440.644,E2 -4440.644} C_VEL
LIN {X 0,Y 530.988,Z 127.343,A -85,B 0,C 180,E1 -4443.772,E2 -4443.772} C_VEL
LIN {X 0,Y 530.956,Z 127.343,A -85,B 0,C 180,E1 -4446.558,E2 -4446.558} C_VEL
LIN {X 0,Y 530.989,Z 127.34,A -85,B 0,C 180,E1 -4449.443,E2 -4449.443} C_VEL
LIN {X 0,Y 530.978,Z 127.34,A -85,B 0,C 180,E1 -4452.456,E2 -4452.456} C_VEL
LIN {X 0,Y 530.983,Z 127.346,A -85,B 0,C 180,E1 -4455.621,E2 -4455.621} C_VEL
LIN {X 0,Y 530.997,Z 127.337,A -85,B 0,C 180,E1 -4458.564,E2 -4458.564} C_VEL
LIN {X 0,Y 530.957,Z 127.349,A -85,B 0,C 180,E1 -4461.529,E2 -4461.529} C_VEL
LIN {X 0,Y 530.953,Z 127.342,A -85,B 0,C 180,E1 -4464.379,E2 -4464.379} C_VEL
LIN {X 0,Y 530.966,Z 127.344,A -85,B 0,C 180,E1 -4467.133,E2 -4467.133} C_VEL
LIN {X 0,Y 530.96,Z 127.345,A -85,B 0,C 180,E1 -4469.802,E2 -4469.802} C_VEL
LIN {X 0,Y 531.012,Z 127.335,A -85,B 0,C 180,E1 -4472.467,E2 -4472.467} C_VEL
LIN {X 0,Y 531.005,Z 127.339,A -85,B 0,C 180,E1 -4474.942,E2 -4474.942} C_VEL
LIN {X 0,Y 530.971,Z 127.34,A -85,B 0,C 180,E1 -4478.246,E2 -4478.246} C_VEL
LIN {X 0,Y 530.991,Z 127.339,A -85,B 0,C 180,E1 -4480.677,E2 -4480.677} C_VEL
LIN {X 0,Y 530.974,Z 127.347,A -85,B 0,C 180,E1 -4483.07,E2 -4483.07} C_VEL
LIN {X 0,Y 531.018,Z 127.339,A -85,B 0,C 180,E1 -4485.435,E2 -4485.435} C_VEL
LIN {X 0,Y 531.036,Z 127.334,A -85,B 0,C 180,E1 -4488.549,E2 -4488.549} C_VEL
LIN {X 0,Y 531.054,Z 127.331,A -85,B 0,C 180,E1 -4491.629,E2 -4491.629} C_VEL
LIN {X 0,Y 531.12,Z 127.326,A -85,B 0,C 180,E1 -4494.685,E2 -4494.685} C_VEL
LIN {X 0,Y 531.14,Z 127.319,A -85,B 0,C 180,E1 -4497.725,E2 -4497.725} C_VEL
LIN {X 0,Y 531.153,Z 127.325,A -85,B 0,C 180,E1 -4500.758,E2 -4500.758} C_VEL
LIN {X 0,Y 531.103,Z 127.329,A -85,B 0,C 180,E1 -4503.034,E2 -4503.034} C_VEL
LIN {X 0,Y 531.075,Z 127.328,A -85,B 0,C 180,E1 -4506.077,E2 -4506.077} C_VEL
LIN {X 0,Y 531.03,Z 127.335,A -85,B 0,C 180,E1 -4509.138,E2 -4509.138} C_VEL
LIN {X 0,Y 531.038,Z 127.335,A -85,B 0,C 180,E1 -4512.225,E2 -4512.225} C_VEL
LIN {X 0,Y 530.993,Z 127.337,A -85,B 0,C 180,E1 -4515.349,E2 -4515.349} C_VEL
LIN {X 0,Y 530.988,Z 127.346,A -85,B 0,C 180,E1 -4518.521,E2 -4518.521} C_VEL
LIN {X 0,Y 530.997,Z 127.339,A -85,B 0,C 180,E1 -4520.938,E2 -4520.938} C_VEL
LIN {X 0,Y 530.969,Z 127.347,A -85,B 0,C 180,E1 -4524.225,E2 -4524.225} C_VEL
LIN {X 0,Y 531.009,Z 127.338,A -85,B 0,C 180,E1 -4526.743,E2 -4526.743} C_VEL
LIN {X 0,Y 530.979,Z 127.339,A -85,B 0,C 180,E1 -4529.322,E2 -4529.322} C_VEL
LIN {X 0,Y 530.977,Z 127.347,A -85,B 0,C 180,E1 -4532.103,E2 -4532.103} C_VEL
LIN {X 0,Y 530.98,Z 127.339,A -85,B 0,C 180,E1 -4534.853,E2 -4534.853} C_VEL
LIN {X 0,Y 530.963,Z 127.342,A -85,B 0,C 180,E1 -4537.507,E2 -4537.507} C_VEL
LIN {X 0,Y 531.022,Z 127.337,A -85,B 0,C 180,E1 -4540.428,E2 -4540.428} C_VEL
LIN {X 0,Y 530.959,Z 127.343,A -85,B 0,C 180,E1 -4543.566,E2 -4543.566} C_VEL
LIN {X 0,Y 530.286,Z 127.431,A -85,B 0,C 180,E1 -4544.199,E2 -4544.199} C_VEL
LIN {X 0,Y 527.439,Z 127.781,A -85,B 0,C 180,E1 -4545.228,E2 -4545.228} C_VEL
LIN {X 0,Y 525.036,Z 128.086,A -85,B 0,C 180,E1 -4546.057,E2 -4546.057} C_VEL
LIN {X 0,Y 524.003,Z 128.209,A -85,B 0,C 180,E1 -4546.696,E2 -4546.696} C_VEL
LIN {X 0,Y 523.918,Z 128.218,A -85,B 0,C 180,E1 -4546.913,E2 -4546.913} C_VEL
LIN {X 0,Y 523.974,Z 128.219,A -85,B 0,C 180,E1 -4549.923,E2 -4549.923} C_VEL
LIN {X 0,Y 523.908,Z 128.22,A -85,B 0,C 180,E1 -4552.868,E2 -4552.868} C_VEL
LIN {X 0,Y 523.936,Z 128.225,A -85,B 0,C 180,E1 -4555.711,E2 -4555.711} C_VEL
LIN {X 0,Y 523.927,Z 128.218,A -85,B 0,C 180,E1 -4558.457,E2 -4558.457} C_VEL
LIN {X 0,Y 523.936,Z 128.219,A -85,B 0,C 180,E1 -4561.126,E2 -4561.126} C_VEL
LIN {X 0,Y 523.98,Z 128.214,A -85,B 0,C 180,E1 -4563.98,E2 -4563.98} C_VEL
LIN {X 0,Y 523.932,Z 128.217,A -85,B 0,C 180,E1 -4566.271,E2 -4566.271} C_VEL
LIN {X 0,Y 523.943,Z 128.216,A -85,B 0,C 180,E1 -4568.767,E2 -4568.767} C_VEL
LIN {X 0,Y 523.948,Z 128.221,A -85,B 0,C 180,E1 -4571.221,E2 -4571.221} C_VEL
LIN {X 0,Y 523.934,Z 128.221,A -85,B 0,C 180,E1 -4573.639,E2 -4573.639} C_VEL
LIN {X 0,Y 523.941,Z 128.216,A -85,B 0,C 180,E1 -4576.028,E2 -4576.028} C_VEL
LIN {X 0,Y 524.008,Z 128.207,A -85,B 0,C 180,E1 -4578.394,E2 -4578.394} C_VEL
LIN {X 0,Y 524.002,Z 128.212,A -85,B 0,C 180,E1 -4581.516,E2 -4581.516} C_VEL
LIN {X 0,Y 524.084,Z 128.2,A -85,B 0,C 180,E1 -4584.614,E2 -4584.614} C_VEL
LIN {X 0,Y 524.111,Z 128.195,A -85,B 0,C 180,E1 -4587.695,E2 -4587.695} C_VEL
LIN {X 0,Y 524.121,Z 128.199,A -85,B 0,C 180,E1 -4590.769,E2 -4590.769} C_VEL
LIN {X 0,Y 524.069,Z 128.207,A -85,B 0,C 180,E1 -4593.075,E2 -4593.075} C_VEL
LIN {X 0,Y 524.051,Z 128.202,A -85,B 0,C 180,E1 -4596.159,E2 -4596.159} C_VEL
LIN {X 0,Y 523.997,Z 128.211,A -85,B 0,C 180,E1 -4599.262,E2 -4599.262} C_VEL
LIN {X 0,Y 524.001,Z 128.208,A -85,B 0,C 180,E1 -4601.74,E2 -4601.74} C_VEL
LIN {X 0,Y 523.992,Z 128.215,A -85,B 0,C 180,E1 -4605.053,E2 -4605.053} C_VEL
LIN {X 0,Y 523.965,Z 128.217,A -85,B 0,C 180,E1 -4607.969,E2 -4607.969} C_VEL
LIN {X 0,Y 524,Z 128.425,A -85,B 0,C 180,E1 -4609.032,E2 -4609.032} C_VEL
LIN {X 0,Y 524.481,Z 132.857,A -85,B 0,C 180,E1 -4609.923,E2 -4609.923} C_VEL
LIN {X 0,Y 524.248,Z 148.147,A -85,B 0,C 180,E1 -4612.905,E2 -4612.905} C_VEL
LIN {X 0,Y 525.988,Z 158.586,A -85,B 0,C 180,E1 -4613.11,E2 -4613.11} C_VEL
LIN {X 0,Y 525.478,Z 254.423,A -85,B 0,C 180,E1 -4614.45,E2 -4614.45} C_VEL
LIN {X 0,Y 525.29,Z 267.433,A -85,B 0,C 180,E1 -4614.78,E2 -4614.78} C_VEL
LIN {X 0,Y 525.141,Z 279.622,A -85,B 0,C 180,E1 -4615.241,E2 -4615.241} C_VEL
LIN {X 0,Y 524.951,Z 290.547,A -85,B 0,C 180,E1 -4615.793,E2 -4615.793} C_VEL
LIN {X 0,Y 524.657,Z 300.852,A -85,B 0,C 180,E1 -4616.449,E2 -4616.449} C_VEL
LIN {X 0,Y 524.379,Z 311.634,A -85,B 0,C 180,E1 -4617.312,E2 -4617.312} C_VEL
LIN {X 0,Y 524.121,Z 321.735,A -85,B 0,C 180,E1 -4618.317,E2 -4618.317} C_VEL
LIN {X 0,Y 523.924,Z 329.93,A -85,B 0,C 180,E1 -4619.319,E2 -4619.319} C_VEL
LIN {X 0,Y 523.72,Z 337.416,A -85,B 0,C 180,E1 -4620.437,E2 -4620.437} C_VEL
LIN {X 0,Y 523.611,Z 343.495,A -85,B 0,C 180,E1 -4621.566,E2 -4621.566} C_VEL
LIN {X 0,Y 523.455,Z 349.277,A -85,B 0,C 180,E1 -4622.941,E2 -4622.941} C_VEL
LIN {X 0,Y 523.383,Z 353.585,A -85,B 0,C 180,E1 -4624.332,E2 -4624.332} C_VEL
LIN {X 0,Y 523.303,Z 355.64,A -85,B 0,C 180,E1 -4625.275,E2 -4625.275} C_VEL
LIN {X 0,Y 523.301,Z 357.22,A -85,B 0,C 180,E1 -4626.313,E2 -4626.313} C_VEL
LIN {X 0,Y 523.248,Z 358.15,A -85,B 0,C 180,E1 -4627.585,E2 -4627.585} C_VEL
LIN {X 0,Y 523.269,Z 357.828,A -85,B 0,C 180,E1 -4629.143,E2 -4629.143} C_VEL
LIN {X 0,Y 523.291,Z 356.763,A -85,B 0,C 180,E1 -4630.141,E2 -4630.141} C_VEL
LIN {X 0,Y 523.383,Z 354.82,A -85,B 0,C 180,E1 -4631.24,E2 -4631.24} C_VEL
LIN {X 0,Y 523.411,Z 351.839,A -85,B 0,C 180,E1 -4632.397,E2 -4632.397} C_VEL
LIN {X 0,Y 523.523,Z 347.877,A -85,B 0,C 180,E1 -4633.539,E2 -4633.539} C_VEL
LIN {X 0,Y 523.608,Z 342.936,A -85,B 0,C 180,E1 -4634.654,E2 -4634.654} C_VEL
LIN {X 0,Y 523.793,Z 336.1,A -85,B 0,C 180,E1 -4635.875,E2 -4635.875} C_VEL
LIN {X 0,Y 523.985,Z 328.076,A -85,B 0,C 180,E1 -4637.026,E2 -4637.026} C_VEL
LIN {X 0,Y 524.233,Z 318.738,A -85,B 0,C 180,E1 -4638.106,E2 -4638.106} C_VEL
LIN {X 0,Y 524.483,Z 308.352,A -85,B 0,C 180,E1 -4639.069,E2 -4639.069} C_VEL
LIN {X 0,Y 524.749,Z 296.855,A -85,B 0,C 180,E1 -4639.922,E2 -4639.922} C_VEL
LIN {X 0,Y 525.081,Z 284.596,A -85,B 0,C 180,E1 -4640.62,E2 -4640.62} C_VEL
LIN {X 0,Y 525.283,Z 272.005,A -85,B 0,C 180,E1 -4641.16,E2 -4641.16} C_VEL
LIN {X 0,Y 525.425,Z 259.208,A -85,B 0,C 180,E1 -4641.54,E2 -4641.54} C_VEL
LIN {X 0,Y 525.568,Z 243.418,A -85,B 0,C 180,E1 -4641.808,E2 -4641.808} C_VEL
LIN {X 0,Y 525.954,Z 156.981,A -85,B 0,C 180,E1 -4643.007,E2 -4643.007} C_VEL
LIN {X 0,Y 524.281,Z 148.237,A -85,B 0,C 180,E1 -4643.197,E2 -4643.197} C_VEL
LIN {X 0,Y 524.422,Z 133.403,A -85,B 0,C 180,E1 -4646.014,E2 -4646.014} C_VEL
LIN {X 0,Y 523.989,Z 128.218,A -85,B 0,C 180,E1 -4647.041,E2 -4647.041} C_VEL
LIN {X 0,Y 523.94,Z 128.218,A -85,B 0,C 180,E1 -4650.245,E2 -4650.245} C_VEL
LIN {X 0,Y 523.95,Z 128.221,A -85,B 0,C 180,E1 -4652.867,E2 -4652.867} C_VEL
LIN {X 0,Y 523.938,Z 128.22,A -85,B 0,C 180,E1 -4655.804,E2 -4655.804} C_VEL
LIN {X 0,Y 523.948,Z 128.222,A -85,B 0,C 180,E1 -4658.767,E2 -4658.767} C_VEL
LIN {X 0,Y 523.941,Z 128.221,A -85,B 0,C 180,E1 -4661.221,E2 -4661.221} C_VEL
LIN {X 0,Y 523.924,Z 128.22,A -85,B 0,C 180,E1 -4663.639,E2 -4663.639} C_VEL
LIN {X 0,Y 523.928,Z 128.22,A -85,B 0,C 180,E1 -4666.028,E2 -4666.028} C_VEL
LIN {X 0,Y 523.996,Z 128.211,A -85,B 0,C 180,E1 -4669.178,E2 -4669.178} C_VEL
LIN {X 0,Y 523.98,Z 128.218,A -85,B 0,C 180,E1 -4672.292,E2 -4672.292} C_VEL
LIN {X 0,Y 524.039,Z 128.21,A -85,B 0,C 180,E1 -4674.614,E2 -4674.614} C_VEL
LIN {X 0,Y 524.108,Z 128.197,A -85,B 0,C 180,E1 -4677.695,E2 -4677.695} C_VEL
LIN {X 0,Y 524.101,Z 128.199,A -85,B 0,C 180,E1 -4680,E2 -4680} C_VEL
LIN {X 0,Y 524.108,Z 128.2,A -85,B 0,C 180,E1 -4682.306,E2 -4682.306} C_VEL
LIN {X 0,Y 524.004,Z 128.212,A -85,B 0,C 180,E1 -4686.16,E2 -4686.16} C_VEL
LIN {X 0,Y 523.947,Z 128.216,A -85,B 0,C 180,E1 -4689.263,E2 -4689.263} C_VEL
LIN {X 0,Y 523.923,Z 128.219,A -85,B 0,C 180,E1 -4692.394,E2 -4692.394} C_VEL
LIN {X 0,Y 523.884,Z 128.227,A -85,B 0,C 180,E1 -4695.564,E2 -4695.564} C_VEL
LIN {X 0,Y 523.89,Z 128.225,A -85,B 0,C 180,E1 -4697.972,E2 -4697.972} C_VEL
LIN {X 0,Y 523.894,Z 128.221,A -85,B 0,C 180,E1 -4700.414,E2 -4700.414} C_VEL
LIN {X 0,Y 523.888,Z 128.225,A -85,B 0,C 180,E1 -4702.895,E2 -4702.895} C_VEL
LIN {X 0,Y 523.879,Z 128.231,A -85,B 0,C 180,E1 -4705.423,E2 -4705.423} C_VEL
LIN {X 0,Y 523.9,Z 128.22,A -85,B 0,C 180,E1 -4708.003,E2 -4708.003} C_VEL
LIN {X 0,Y 523.902,Z 128.226,A -85,B 0,C 180,E1 -4710.846,E2 -4710.846} C_VEL
LIN {X 0,Y 523.931,Z 128.218,A -85,B 0,C 180,E1 -4713.729,E2 -4713.729} C_VEL
LIN {X 0,Y 523.902,Z 128.223,A -85,B 0,C 180,E1 -4716.4,E2 -4716.4} C_VEL
LIN {X 0,Y 523.916,Z 128.225,A -85,B 0,C 180,E1 -4719.086,E2 -4719.086} C_VEL
LIN {X 0,Y 523.904,Z 128.222,A -85,B 0,C 180,E1 -4722.124,E2 -4722.124} C_VEL
LIN {X 0,Y 523.941,Z 128.219,A -85,B 0,C 180,E1 -4725.311,E2 -4725.311} C_VEL
LIN {X 0,Y 523.944,Z 128.223,A -85,B 0,C 180,E1 -4728.692,E2 -4728.692} C_VEL
LIN {X 0,Y 523.917,Z 128.223,A -85,B 0,C 180,E1 -4731.898,E2 -4731.898} C_VEL
LIN {X 0,Y 523.928,Z 128.22,A -85,B 0,C 180,E1 -4734.911,E2 -4734.911} C_VEL
LIN {X 0,Y 523.94,Z 128.222,A -85,B 0,C 180,E1 -4737.68,E2 -4737.68} C_VEL
LIN {X 0,Y 523.957,Z 128.217,A -85,B 0,C 180,E1 -4740.677,E2 -4740.677} C_VEL
LIN {X 0,Y 523.941,Z 128.223,A -85,B 0,C 180,E1 -4743.726,E2 -4743.726} C_VEL
LIN {X 0,Y 524.022,Z 128.338,A -85,B 0,C 180,E1 -4745.194,E2 -4745.194} C_VEL
LIN {X 0,Y 525.353,Z 136.817,A -85,B 0,C 180,E1 -4746.547,E2 -4746.547} C_VEL
LIN {X 0,Y 524.845,Z 158.676,A -85,B 0,C 180,E1 -4749.829,E2 -4749.829} C_VEL
LIN {X 0,Y 524.522,Z 177.718,A -85,B 0,C 180,E1 -4752.655,E2 -4752.655} C_VEL
LIN {X 0,Y 524.198,Z 192.51,A -85,B 0,C 180,E1 -4754.826,E2 -4754.826} C_VEL
LIN {X 0,Y 525.878,Z 204.351,A -85,B 0,C 180,E1 -4755.053,E2 -4755.053} C_VEL
LIN {X 0,Y 525.468,Z 301.5,A -85,B 0,C 180,E1 -4756.414,E2 -4756.414} C_VEL
LIN {X 0,Y 525.224,Z 314.704,A -85,B 0,C 180,E1 -4756.753,E2 -4756.753} C_VEL
LIN {X 0,Y 524.947,Z 327.423,A -85,B 0,C 180,E1 -4757.238,E2 -4757.238} C_VEL
LIN {X 0,Y 524.679,Z 339.495,A -85,B 0,C 180,E1 -4757.867,E2 -4757.867} C_VEL
LIN {X 0,Y 524.389,Z 351.743,A -85,B 0,C 180,E1 -4758.696,E2 -4758.696} C_VEL
LIN {X 0,Y 524.13,Z 362.038,A -85,B 0,C 180,E1 -4759.57,E2 -4759.57} C_VEL
LIN {X 0,Y 523.918,Z 371.29,A -85,B 0,C 180,E1 -4760.541,E2 -4760.541} C_VEL
LIN {X 0,Y 523.675,Z 380.298,A -85,B 0,C 180,E1 -4761.704,E2 -4761.704} C_VEL
LIN {X 0,Y 523.569,Z 387.557,A -85,B 0,C 180,E1 -4762.867,E2 -4762.867} C_VEL
LIN {X 0,Y 523.458,Z 392.451,A -85,B 0,C 180,E1 -4763.834,E2 -4763.834} C_VEL
LIN {X 0,Y 523.383,Z 397.211,A -85,B 0,C 180,E1 -4764.992,E2 -4764.992} C_VEL
LIN {X 0,Y 523.443,Z 400.853,A -85,B 0,C 180,E1 -4766.15,E2 -4766.15} C_VEL
LIN {X 0,Y 523.391,Z 402.729,A -85,B 0,C 180,E1 -4766.921,E2 -4766.921} C_VEL
LIN {X 0,Y 523.337,Z 404.135,A -85,B 0,C 180,E1 -4767.691,E2 -4767.691} C_VEL
LIN {X 0,Y 523.263,Z 405.753,A -85,B 0,C 180,E1 -4769.23,E2 -4769.23} C_VEL
LIN {X 0,Y 523.265,Z 405.974,A -85,B 0,C 180,E1 -4770,E2 -4770} C_VEL
LIN {X 0,Y 523.275,Z 405.152,A -85,B 0,C 180,E1 -4771.539,E2 -4771.539} C_VEL
LIN {X 0,Y 523.337,Z 404.157,A -85,B 0,C 180,E1 -4772.308,E2 -4772.308} C_VEL
LIN {X 0,Y 523.391,Z 402.758,A -85,B 0,C 180,E1 -4773.078,E2 -4773.078} C_VEL
LIN {X 0,Y 523.422,Z 399.811,A -85,B 0,C 180,E1 -4774.235,E2 -4774.235} C_VEL
LIN {X 0,Y 523.455,Z 395.818,A -85,B 0,C 180,E1 -4775.392,E2 -4775.392} C_VEL
LIN {X 0,Y 523.507,Z 389.728,A -85,B 0,C 180,E1 -4776.735,E2 -4776.735} C_VEL
LIN {X 0,Y 523.643,Z 382.961,A -85,B 0,C 180,E1 -4777.907,E2 -4777.907} C_VEL
LIN {X 0,Y 523.819,Z 374.633,A -85,B 0,C 180,E1 -4779.07,E2 -4779.07} C_VEL
LIN {X 0,Y 524.014,Z 366.088,A -85,B 0,C 180,E1 -4780.041,E2 -4780.041} C_VEL
LIN {X 0,Y 524.295,Z 355.535,A -85,B 0,C 180,E1 -4781.012,E2 -4781.012} C_VEL
LIN {X 0,Y 524.581,Z 343.649,A -85,B 0,C 180,E1 -4781.887,E2 -4781.887} C_VEL
LIN {X 0,Y 524.872,Z 331.675,A -85,B 0,C 180,E1 -4782.567,E2 -4782.567} C_VEL
LIN {X 0,Y 525.128,Z 319.211,A -85,B 0,C 180,E1 -4783.101,E2 -4783.101} C_VEL
LIN {X 0,Y 525.363,Z 306.322,A -85,B 0,C 180,E1 -4783.489,E2 -4783.489} C_VEL
LIN {X 0,Y 525.531,Z 290.856,A -85,B 0,C 180,E1 -4783.756,E2 -4783.756} C_VEL
LIN {X 0,Y 525.735,Z 203.056,A -85,B 0,C 180,E1 -4784.972,E2 -4784.972} C_VEL
LIN {X 0,Y 524.228,Z 192.805,A -85,B 0,C 180,E1 -4785.174,E2 -4785.174} C_VEL
LIN {X 0,Y 524.627,Z 173.855,A -85,B 0,C 180,E1 -4787.986,E2 -4787.986} C_VEL
LIN {X 0,Y 525.099,Z 152.561,A -85,B 0,C 180,E1 -4791.184,E2 -4791.184} C_VEL
LIN {X 0,Y 525.508,Z 136.374,A -85,B 0,C 180,E1 -4793.653,E2 -4793.653} C_VEL
LIN {X 0,Y 523.977,Z 128.217,A -85,B 0,C 180,E1 -4794.992,E2 -4794.992} C_VEL
LIN {X 0,Y 523.958,Z 128.222,A -85,B 0,C 180,E1 -4797.999,E2 -4797.999} C_VEL
LIN {X 0,Y 523.946,Z 128.216,A -85,B 0,C 180,E1 -4800.854,E2 -4800.854} C_VEL
LIN {X 0,Y 523.96,Z 128.218,A -85,B 0,C 180,E1 -4803.734,E2 -4803.734} C_VEL
LIN {X 0,Y 523.904,Z 128.223,A -85,B 0,C 180,E1 -4806.401,E2 -4806.401} C_VEL
LIN {X 0,Y 523.922,Z 128.218,A -85,B 0,C 180,E1 -4809.084,E2 -4809.084} C_VEL
LIN {X 0,Y 523.952,Z 128.219,A -85,B 0,C 180,E1 -4812.118,E2 -4812.118} C_VEL
LIN {X 0,Y 523.946,Z 128.218,A -85,B 0,C 180,E1 -4815.309,E2 -4815.309} C_VEL
LIN {X 0,Y 523.958,Z 128.213,A -85,B 0,C 180,E1 -4818.689,E2 -4818.689} C_VEL
LIN {X 0,Y 523.917,Z 128.22,A -85,B 0,C 180,E1 -4821.08,E2 -4821.08} C_VEL
LIN {X 0,Y 523.9,Z 128.226,A -85,B 0,C 180,E1 -4823.825,E2 -4823.825} C_VEL
LIN {X 0,Y 523.912,Z 128.219,A -85,B 0,C 180,E1 -4826.633,E2 -4826.633} C_VEL
LIN {X 0,Y 523.948,Z 128.222,A -85,B 0,C 180,E1 -4829.355,E2 -4829.355} C_VEL
LIN {X 0,Y 523.976,Z 128.211,A -85,B 0,C 180,E1 -4832.281,E2 -4832.281} C_VEL
LIN {X 0,Y 523.952,Z 128.214,A -85,B 0,C 180,E1 -4834.581,E2 -4834.581} C_VEL
LIN {X 0,Y 523.911,Z 128.225,A -85,B 0,C 180,E1 -4837.106,E2 -4837.106} C_VEL
LIN {X 0,Y 523.978,Z 128.212,A -85,B 0,C 180,E1 -4839.866,E2 -4839.866} C_VEL
LIN {X 0,Y 523.956,Z 128.217,A -85,B 0,C 180,E1 -4842.836,E2 -4842.836} C_VEL
LIN {X 0,Y 523.976,Z 128.219,A -85,B 0,C 180,E1 -4845.235,E2 -4845.235} C_VEL
LIN {X 0,Y 524.011,Z 128.208,A -85,B 0,C 180,E1 -4848.394,E2 -4848.394} C_VEL
LIN {X 0,Y 524.002,Z 128.21,A -85,B 0,C 180,E1 -4851.516,E2 -4851.516} C_VEL
LIN {X 0,Y 524.081,Z 128.202,A -85,B 0,C 180,E1 -4854.613,E2 -4854.613} C_VEL
LIN {X 0,Y 524.112,Z 128.195,A -85,B 0,C 180,E1 -4857.694,E2 -4857.694} C_VEL
LIN {X 0,Y 524.123,Z 128.201,A -85,B 0,C 180,E1 -4860.768,E2 -4860.768} C_VEL
LIN {X 0,Y 524.069,Z 128.204,A -85,B 0,C 180,E1 -4863.074,E2 -4863.074} C_VEL
LIN {X 0,Y 524.036,Z 128.205,A -85,B 0,C 180,E1 -4866.159,E2 -4866.159} C_VEL
LIN {X 0,Y 524.002,Z 128.214,A -85,B 0,C 180,E1 -4868.484,E2 -4868.484} C_VEL
LIN {X 0,Y 524.001,Z 128.208,A -85,B 0,C 180,E1 -4871.739,E2 -4871.739} C_VEL
LIN {X 0,Y 523.991,Z 128.211,A -85,B 0,C 180,E1 -4875.052,E2 -4875.052} C_VEL
